  MoveC 2658 to (-287.4, 215.34, -30) mm, rotated rx 180 ry 0 rz 0.01 deg; joints [34.37, -40.028, 93.325, -139.792, 61.018, 158.683] to (-287.36, 219.75, -30) mm, rotated rx -180 ry 0 rz 0.01 deg; joints [34.501, -39.911, 93.073, -139.606, 60.965, 158.515]
  MoveC 2659 to (-287.18, 224.12, -30) mm, rotated rx 180 ry 0 rz 0.01 deg; joints [34.632, -39.801, 92.835, -139.421, 60.919, 158.351] to (-289.23, 227.97, -30) mm, rotated rx 180 ry 0 rz 0.01 deg; joints [34.703, -39.613, 92.434, -139.269, 60.786, 158.156]
  MoveC 2660 to (-302.15, 245.09, -30) mm, rotated rx -180 ry 0 rz 0.01 deg; joints [34.939, -38.61, 90.306, -138.602, 60.033, 157.181] to (-311.06, 264.6, -30) mm, rotated rx 180 ry 0 rz 0.01 deg; joints [35.316, -37.679, 88.333, -137.799, 59.413, 156.172]
  MoveC 2661 to (-313.16, 267.48, -30) mm, rotated rx -180 ry 0 rz 0.01 deg; joints [35.355, -37.507, 87.968, -137.682, 59.287, 156] to (-316.55, 268.57, -30) mm, rotated rx 180 ry 0 rz 0.01 deg; joints [35.318, -37.331, 87.599, -137.643, 59.129, 155.869]
  MoveL 2662 to (-329.31, 268.57, -30) mm, rotated rx 180 ry 0 rz 0.01 deg; joints [35.065, -36.784, 86.459, -137.668, 58.581, 155.543]
  MoveC 2663 to (-332.03, 267.45, -30) mm, rotated rx 180 ry 0 rz 0.01 deg; joints [34.98, -36.7, 86.285, -137.721, 58.477, 155.52] to (-333.16, 264.72, -30) mm, rotated rx 180 ry 0 rz 0.01 deg; joints [34.881, -36.731, 86.354, -137.84, 58.463, 155.605]
  MoveL 2664 to (-333.15, 129.67, -30) mm, rotated rx -180 ry 0 rz 0.01 deg; joints [30.91, -40.332, 94.104, -143.652, 60.117, 160.875]
  MoveC 2665 to (-332.02, 125.86, -30) mm, rotated rx -180 ry 0 rz 0.01 deg; joints [30.814, -40.47, 94.4, -143.81, 60.211, 161.035] to (-328.98, 123.31, -30) mm, rotated rx 180 ry 0 rz 0.01 deg; joints [30.791, -40.656, 94.796, -143.905, 60.373, 161.19]
  MoveC 2666 to (-314.64, 115.76, -30) mm, rotated rx 180 ry 0 rz 0.01 deg; joints [30.822, -41.42, 96.418, -144.154, 61.078, 161.751] to (-301.61, 106.12, -30) mm, rotated rx -180 ry 0 rz 0.01 deg; joints [30.764, -42.166, 98.01, -144.486, 61.745, 162.344]
  MoveC 2667 to (-290.27, 94.52, -30) mm, rotated rx -180 ry 0 rz 0.01 deg; joints [30.609, -42.877, 99.534, -144.901, 62.359, 162.955] to (-281.02, 81.2, -30) mm, rotated rx 180 ry 0 rz 0.01 deg; joints [30.356, -43.533, 100.948, -145.396, 62.903, 163.57]
  MoveL 2668 to (-263.17, 49.55, -30) mm, rotated rx 180 ry 0 rz 0.01 deg; joints [29.657, -44.892, 103.897, -146.586, 64.014, 164.905]
  MoveC 2669 to (-262.35, 48.05, -30) mm, rotated rx -180 ry 0 rz 0.01 deg; joints [29.623, -44.954, 104.032, -146.643, 64.065, 164.966] to (-261.62, 46.51, -30) mm, rotated rx -180 ry 0 rz 0.01 deg; joints [29.585, -45.014, 104.161, -146.702, 64.114, 165.027]
  MoveC 2670 to (-260.93, 44.95, -30) mm, rotated rx 180 ry 0 rz 0.01 deg; joints [29.546, -45.072, 104.289, -146.762, 64.16, 165.088] to (-260.22, 43.39, -30) mm, rotated rx -180 ry 0 rz 0.01 deg; joints [29.508, -45.131, 104.417, -146.821, 64.208, 165.148]
  MoveC 2671 to (-257.67, 40.46, -30) mm, rotated rx -180 ry 0 rz 0.01 deg; joints [29.458, -45.287, 104.757, -146.922, 64.347, 165.283] to (-253.93, 39.36, -30) mm, rotated rx -180 ry 0 rz 0.01 deg; joints [29.492, -45.45, 105.107, -146.935, 64.514, 165.38]
  MoveL 2672 to (-139.56, 39.36, -30) mm, rotated rx -180 ry 0 rz 0.01 deg; joints [31.818, -49.526, 113.886, -145.611, 69.031, 167.233]
  MoveC 2673 to (-135.82, 40.46, -30) mm, rotated rx 180 ry 0 rz 0.01 deg; joints [31.938, -49.631, 114.111, -145.512, 69.16, 167.26] to (-133.27, 43.42, -30) mm, rotated rx 180 ry 0 rz 0.01 deg; joints [32.098, -49.657, 114.162, -145.351, 69.219, 167.214]
  MoveC 2674 to (-132.52, 45.08, -30) mm, rotated rx 180 ry 0 rz 0.01 deg; joints [32.173, -49.649, 114.141, -145.271, 69.227, 167.178] to (-131.78, 46.75, -30) mm, rotated rx 180 ry 0 rz 0.01 deg; joints [32.247, -49.64, 114.118, -145.191, 69.234, 167.141]
  MoveC 2675 to (-131.01, 48.4, -30) mm, rotated rx -180 ry 0 rz 0.01 deg; joints [32.322, -49.633, 114.099, -145.11, 69.242, 167.106] to (-130.14, 50, -30) mm, rotated rx -180 ry 0 rz 0.01 deg; joints [32.397, -49.629, 114.088, -145.031, 69.255, 167.073]
  MoveL 2676 to (-112.26, 81.56, -30) mm, rotated rx -180 ry 0 rz 0.01 deg; joints [33.893, -49.569, 113.893, -143.455, 69.523, 166.428]
  MoveC 2677 to (-103.05, 94.8, -30) mm, rotated rx 180 ry 0 rz 0.01 deg; joints [34.56, -49.588, 113.908, -142.767, 69.693, 166.179] to (-91.75, 106.32, -30) mm, rotated rx 180 ry 0 rz 0.01 deg; joints [35.217, -49.706, 114.14, -142.117, 69.958, 166.013]
  MoveC 2678 to (-78.77, 115.88, -30) mm, rotated rx 180 ry 0 rz 0.01 deg; joints [35.853, -49.913, 114.573, -141.516, 70.303, 165.933] to (-64.48, 123.34, -30) mm, rotated rx 180 ry 0 rz 0.01 deg; joints [36.455, -50.202, 115.186, -140.973, 70.717, 165.937]
  MoveC 2679 to (-61.48, 125.84, -30) mm, rotated rx 180 ry 0 rz 0.01 deg; joints [36.613, -50.24, 115.265, -140.82, 70.791, 165.909] to (-60.36, 129.58, -30) mm, rotated rx 180 ry 0 rz 0.01 deg; joints [36.767, -50.191, 115.151, -140.649, 70.781, 165.812]
  MoveL 2680 to (-60.36, 264.73, -30) mm, rotated rx -180 ry 0 rz 0.01 deg; joints [41.026, -46.847, 107.689, -135.318, 69.022, 161.344]
  MoveC 2681 to (-61.49, 267.45, -30) mm, rotated rx 180 ry 0 rz 0.01 deg; joints [41.077, -46.737, 107.45, -135.232, 68.948, 161.227] to (-64.21, 268.58, -30) mm, rotated rx 180 ry 0 rz 0.01 deg; joints [41.041, -46.62, 107.197, -135.232, 68.838, 161.138]
  MoveL 2682 to (-76.96, 268.58, -30) mm, rotated rx 180 ry 0 rz 0.01 deg; joints [40.715, -46.209, 106.319, -135.431, 68.393, 160.909]
  MoveC 2683 to (-80.35, 267.48, -30) mm, rotated rx -180 ry 0 rz 0.01 deg; joints [40.597, -46.129, 106.149, -135.525, 68.288, 160.886] to (-82.45, 264.61, -30) mm, rotated rx -180 ry 0 rz 0.01 deg; joints [40.459, -46.138, 106.174, -135.668, 68.25, 160.951]
  MoveC 2684 to (-94.52, 240.3, -30) mm, rotated rx -180 ry 0 rz 0.01 deg; joints [39.431, -46.39, 106.752, -136.798, 68.133, 161.591] to (-112.91, 220.34, -30) mm, rotated rx -180 ry 0 rz 0.01 deg; joints [38.375, -46.299, 106.59, -137.853, 67.726, 161.954]
  MoveC 2685 to (-135.88, 205.99, -30) mm, rotated rx 180 ry 0 rz 0.01 deg; joints [37.386, -45.887, 105.736, -138.74, 67.068, 162.034] to (-161.71, 197.84, -30) mm, rotated rx -180 ry 0 rz 0.01 deg; joints [36.537, -45.199, 104.282, -139.395, 66.206, 161.843]
  MoveC 2686 to (-174.93, 196.15, -30) mm, rotated rx 180 ry 0 rz 0.01 deg; joints [36.185, -44.775, 103.382, -139.62, 65.727, 161.656] to (-188.26, 195.83, -30) mm, rotated rx 180 ry 0 rz 0.01 deg; joints [35.878, -44.307, 102.387, -139.783, 65.221, 161.417]
  MoveC 2687 to (-201.58, 196.1, -30) mm, rotated rx 180 ry 0 rz 0.01 deg; joints [35.593, -43.817, 101.348, -139.912, 64.703, 161.154] to (-214.9, 196.19, -30) mm, rotated rx -180 ry 0 rz 0.01 deg; joints [35.307, -43.325, 100.306, -140.04, 64.182, 160.893]
  MoveC 2688 to (-245.9, 200.97, -30) mm, rotated rx 180 ry 0 rz 0.01 deg; joints [34.794, -42.036, 97.572, -140.115, 62.891, 160.102] to (-274.04, 214.84, -30) mm, rotated rx 180 ry 0 rz 0.01 deg; joints [34.626, -40.576, 94.475, -139.736, 61.577, 158.995]
  MoveC 2689 to (-281.97, 221.02, -30) mm, rotated rx 180 ry 0 rz 0.01 deg; joints [34.647, -40.094, 93.454, -139.523, 61.173, 158.586] to (-289.23, 227.97, -30) mm, rotated rx 180 ry 0 rz 0.01 deg; joints [34.703, -39.613, 92.434, -139.269, 60.786, 158.156]
  MoveC 2690 to (-291.33, 232.25, -30) mm, rotated rx -180 ry 0 rz 0.01 deg; joints [34.785, -39.411, 92.003, -139.099, 60.646, 157.941] to (-290.67, 236.97, -30) mm, rotated rx 180 ry 0 rz 0.01 deg; joints [34.936, -39.307, 91.78, -138.897, 60.615, 157.771]
  MoveC 2691 to (-289.84, 241.61, -30) mm, rotated rx -180 ry 0 rz 0.01 deg; joints [35.087, -39.213, 91.574, -138.697, 60.592, 157.608] to (-291.43, 246.05, -30) mm, rotated rx -180 ry 0 rz 0.01 deg; joints [35.182, -39.024, 91.172, -138.517, 60.47, 157.395]
  MoveC 2692 to (-298.95, 259.4, -30) mm, rotated rx 180 ry 0 rz 0.01 deg; joints [35.412, -38.336, 89.712, -137.981, 59.989, 156.681] to (-303.93, 273.9, -30) mm, rotated rx -180 ry 0 rz 0.01 deg; joints [35.721, -37.707, 88.377, -137.381, 59.598, 155.964]
  MoveC 2693 to (-305.81, 276.81, -30) mm, rotated rx -180 ry 0 rz 0.01 deg; joints [35.765, -37.543, 88.029, -137.262, 59.482, 155.797] to (-309.08, 277.94, -30) mm, rotated rx 180 ry 0 rz 0.01 deg; joints [35.73, -37.371, 87.669, -137.222, 59.329, 155.667]
  MoveL 2694 to (-338.67, 277.94, -30) mm, rotated rx 180 ry 0 rz 0.01 deg; joints [35.143, -36.096, 85.013, -137.269, 58.056, 154.896]
  MoveC 2695 to (-341.39, 276.81, -30) mm, rotated rx -180 ry 0 rz 0.01 deg; joints [35.058, -36.01, 84.836, -137.32, 57.951, 154.872] to (-342.52, 274.08, -30) mm, rotated rx -180 ry 0 rz 0.01 deg; joints [34.96, -36.043, 84.907, -137.44, 57.936, 154.959]
  MoveL 2696 to (-342.52, 123.04, -30) mm, rotated rx -180 ry 0 rz 0.01 deg; joints [30.536, -40.1, 93.628, -143.974, 59.789, 160.915]
  MoveC 2697 to (-341.43, 119.51, -30) mm, rotated rx -180 ry 0 rz 0.01 deg; joints [30.447, -40.229, 93.906, -144.121, 59.878, 161.066] to (-338.54, 117.21, -30) mm, rotated rx 180 ry 0 rz 0.01 deg; joints [30.428, -40.404, 94.278, -144.208, 60.031, 161.209]
  MoveC 2698 to (-329.79, 113.4, -30) mm, rotated rx 180 ry 0 rz 0.01 deg; joints [30.469, -40.856, 95.234, -144.332, 60.456, 161.526] to (-321.33, 108.99, -30) mm, rotated rx -180 ry 0 rz 0.01 deg; joints [30.487, -41.305, 96.188, -144.478, 60.872, 161.853]
  MoveC 2699 to (-313.31, 103.8, -30) mm, rotated rx 180 ry 0 rz 0.01 deg; joints [30.472, -41.75, 97.135, -144.654, 61.276, 162.194] to (-305.96, 97.7, -30) mm, rotated rx -180 ry 0 rz 0.01 deg; joints [30.416, -42.184, 98.062, -144.87, 61.66, 162.547]
  MoveC 2700 to (-295.26, 85.95, -30) mm, rotated rx 180 ry 0 rz 0.01 deg; joints [30.241, -42.872, 99.537, -145.298, 62.251, 163.148] to (-286.59, 72.62, -30) mm, rotated rx -180 ry 0 rz 0.01 deg; joints [29.974, -43.503, 100.899, -145.8, 62.771, 163.749]
  MoveL 2701 to (-271.14, 44.96, -30) mm, rotated rx -180 ry 0 rz 0.01 deg; joints [29.355, -44.683, 103.46, -146.848, 63.738, 164.911]
  MoveC 2702 to (-269.76, 42.31, -30) mm, rotated rx -180 ry 0 rz 0.01 deg; joints [29.292, -44.79, 103.693, -146.949, 63.826, 165.018] to (-268.6, 39.56, -30) mm, rotated rx 180 ry 0 rz 0.01 deg; joints [29.222, -44.891, 103.913, -147.055, 63.907, 165.124]
  MoveC 2703 to (-267.53, 36.78, -30) mm, rotated rx -180 ry 0 rz 0.01 deg; joints [29.149, -44.988, 104.126, -147.164, 63.983, 165.229] to (-266.4, 34.01, -30) mm, rotated rx -180 ry 0 rz 0.01 deg; joints [29.078, -45.087, 104.342, -147.271, 64.062, 165.334]
  MoveC 2704 to (-263.99, 31.09, -30) mm, rotated rx -180 ry 0 rz 0.01 deg; joints [29.025, -45.237, 104.669, -147.374, 64.196, 165.465] to (-260.37, 30, -30) mm, rotated rx 180 ry 0 rz 0.01 deg; joints [29.056, -45.396, 105.01, -147.389, 64.358, 165.56]
  MoveL 2705 to (-133.13, 30, -30) mm, rotated rx -180 ry 0 rz 0.01 deg; joints [31.628, -49.928, 114.781, -145.913, 69.393, 167.601]
  MoveC 2706 to (-129.52, 31.09, -30) mm, rotated rx 180 ry 0 rz 0.01 deg; joints [31.745, -50.028, 114.996, -145.815, 69.516, 167.626] to (-127.12, 33.98, -30) mm, rotated rx 180 ry 0 rz 0.01 deg; joints [31.901, -50.051, 115.04, -145.659, 69.571, 167.581]
  MoveC 2707 to (-125.94, 36.86, -30) mm, rotated rx 180 ry 0 rz 0.01 deg; joints [32.029, -50.033, 114.995, -145.52, 69.579, 167.517] to (-124.82, 39.77, -30) mm, rotated rx -180 ry 0 rz 0.01 deg; joints [32.156, -50.013, 114.944, -145.382, 69.584, 167.451]
  MoveC 2708 to (-123.61, 42.64, -30) mm, rotated rx 180 ry 0 rz 0.01 deg; joints [32.284, -49.996, 114.901, -145.244, 69.594, 167.388] to (-122.17, 45.4, -30) mm, rotated rx -180 ry 0 rz 0.01 deg; joints [32.413, -49.988, 114.879, -145.107, 69.613, 167.331]
  MoveL 2709 to (-103.15, 78.32, -30) mm, rotated rx 180 ry 0 rz 0.01 deg; joints [33.993, -49.937, 114.701, -143.449, 69.902, 166.67]
  MoveC 2710 to (-91.63, 93.87, -30) mm, rotated rx -180 ry 0 rz 0.01 deg; joints [34.797, -49.981, 114.763, -142.626, 70.123, 166.391] to (-76.92, 106.43, -30) mm, rotated rx 180 ry 0 rz 0.01 deg; joints [35.578, -50.181, 115.174, -141.871, 70.493, 166.25]
  MoveC 2711 to (-71.7, 109.64, -30) mm, rotated rx 180 ry 0 rz 0.01 deg; joints [35.814, -50.277, 115.377, -141.653, 70.638, 166.237] to (-66.23, 112.38, -30) mm, rotated rx 180 ry 0 rz 0.01 deg; joints [36.042, -50.39, 115.619, -141.448, 70.798, 166.242]
  MoveC 2712 to (-60.63, 114.83, -30) mm, rotated rx 180 ry 0 rz 0.01 deg; joints [36.263, -50.513, 115.882, -141.252, 70.966, 166.258] to (-54.97, 117.16, -30) mm, rotated rx 180 ry 0 rz 0.01 deg; joints [36.483, -50.639, 116.152, -141.059, 71.136, 166.279]
  MoveC 2713 to (-52.08, 119.49, -30) mm, rotated rx 180 ry 0 rz 0.01 deg; joints [36.635, -50.678, 116.232, -140.913, 71.207, 166.255] to (-50.99, 123.04, -30) mm, rotated rx 180 ry 0 rz 0.01 deg; joints [36.782, -50.632, 116.126, -140.75, 71.198, 166.164]
  MoveL 2714 to (-51, 274.09, -30) mm, rotated rx 180 ry 0 rz 0.01 deg; joints [41.545, -46.89, 107.767, -134.806, 69.225, 161.178]
  MoveC 2715 to (-52.13, 276.81, -30) mm, rotated rx 180 ry 0 rz 0.01 deg; joints [41.596, -46.781, 107.527, -134.72, 69.151, 161.061] to (-54.85, 277.94, -30) mm, rotated rx 180 ry 0 rz 0.01 deg; joints [41.558, -46.663, 107.275, -134.721, 69.043, 160.972]
  MoveL 2716 to (-84.48, 277.94, -30) mm, rotated rx -180 ry 0 rz 0.01 deg; joints [40.8, -45.709, 105.236, -135.182, 68.009, 160.435]
  MoveC 2717 to (-87.74, 276.81, -30) mm, rotated rx -180 ry 0 rz 0.01 deg; joints [40.684, -45.633, 105.077, -135.274, 67.908, 160.416] to (-89.59, 273.9, -30) mm, rotated rx 180 ry 0 rz 0.01 deg; joints [40.553, -45.652, 105.121, -135.414, 67.879, 160.487]
  MoveC 2718 to (-96.46, 255.09, -30) mm, rotated rx 180 ry 0 rz 0.01 deg; joints [39.826, -45.935, 105.754, -136.247, 67.875, 161.035] to (-107.51, 238.41, -30) mm, rotated rx -180 ry 0 rz 0.01 deg; joints [39.054, -46.01, 105.942, -137.062, 67.691, 161.423]
  MoveC 2719 to (-122.04, 224.65, -30) mm, rotated rx -180 ry 0 rz 0.01 deg; joints [38.286, -45.881, 105.689, -137.809, 67.339, 161.64] to (-139.21, 214.4, -30) mm, rotated rx 180 ry 0 rz 0.01 deg; joints [37.566, -45.56, 105.022, -138.447, 66.838, 161.683]
  MoveC 2720 to (-148.66, 210.65, -30) mm, rotated rx 180 ry 0 rz 0.01 deg; joints [37.231, -45.33, 104.538, -138.719, 66.534, 161.64] to (-158.44, 207.86, -30) mm, rotated rx 180 ry 0 rz 0.01 deg; joints [36.919, -45.06, 103.969, -138.952, 66.204, 161.556]
  MoveC 2721 to (-168.46, 206.14, -30) mm, rotated rx -180 ry 0 rz 0.01 deg; joints [36.638, -44.752, 103.316, -139.141, 65.847, 161.429] to (-178.62, 205.56, -30) mm, rotated rx -180 ry 0 rz 0.01 deg; joints [36.391, -44.406, 102.582, -139.281, 65.469, 161.259]
  MoveL 2722 to (-217.27, 205.67, -30) mm, rotated rx -180 ry 0 rz 0.01 deg; joints [35.543, -42.995, 99.591, -139.675, 63.971, 160.508]
  MoveC 2723 to (-236.59, 208, -30) mm, rotated rx 180 ry 0 rz 0.01 deg; joints [35.201, -42.209, 97.926, -139.749, 63.177, 160.035] to (-254.87, 214.67, -30) mm, rotated rx 180 ry 0 rz 0.01 deg; joints [35.016, -41.332, 96.068, -139.615, 62.361, 159.411]
  MoveC 2724 to (-271.59, 225.24, -30) mm, rotated rx 180 ry 0 rz 0.01 deg; joints [34.983, -40.394, 94.078, -139.286, 61.549, 158.654] to (-285.91, 238.89, -30) mm, rotated rx -180 ry 0 rz 0.01 deg; joints [35.088, -39.448, 92.07, -138.792, 60.789, 157.805]
  MoveC 2725 to (-288.76, 242.4, -30) mm, rotated rx 180 ry 0 rz 0.01 deg; joints [35.131, -39.235, 91.618, -138.658, 60.627, 157.602] to (-291.43, 246.05, -30) mm, rotated rx -180 ry 0 rz 0.01 deg; joints [35.182, -39.024, 91.172, -138.517, 60.47, 157.395]
  MoveC 2726 to (-292.73, 250.22, -30) mm, rotated rx -180 ry 0 rz 0.01 deg; joints [35.276, -38.853, 90.808, -138.346, 60.364, 157.199] to (-291.43, 254.39, -30) mm, rotated rx 180 ry 0 rz 0.01 deg; joints [35.421, -38.788, 90.666, -138.164, 60.366, 157.062]
  MoveC 2727 to (-289.96, 258.45, -30) mm, rotated rx 180 ry 0 rz 0.01 deg; joints [35.567, -38.733, 90.544, -137.986, 60.377, 156.934] to (-290.67, 262.7, -30) mm, rotated rx 180 ry 0 rz 0.01 deg; joints [35.674, -38.582, 90.222, -137.809, 60.294, 156.746]
  MoveC 2728 to (-292.97, 268.55, -30) mm, rotated rx 180 ry 0 rz 0.01 deg; joints [35.793, -38.319, 89.662, -137.57, 60.125, 156.453] to (-294.74, 274.58, -30) mm, rotated rx 180 ry 0 rz 0.01 deg; joints [35.927, -38.07, 89.133, -137.321, 59.975, 156.162]
  MoveC 2729 to (-295.23, 276.75, -30) mm, rotated rx -180 ry 0 rz 0.01 deg; joints [35.978, -37.986, 88.955, -137.23, 59.928, 156.061] to (-295.64, 278.92, -30) mm, rotated rx 180 ry 0 rz 0.01 deg; joints [36.031, -37.905, 88.782, -137.139, 59.883, 155.961]
  MoveC 2730 to (-296.04, 281.1, -30) mm, rotated rx 180 ry 0 rz 0.01 deg; joints [36.084, -37.824, 88.61, -137.048, 59.839, 155.861] to (-296.5, 283.27, -30) mm, rotated rx -180 ry 0 rz 0.01 deg; joints [36.135, -37.741, 88.433, -136.957, 59.793, 155.759]
  MoveC 2731 to (-298.31, 286.17, -30) mm, rotated rx -180 ry 0 rz 0.01 deg; joints [36.179, -37.579, 88.091, -136.839, 59.68, 155.593] to (-301.53, 287.3, -30) mm, rotated rx 180 ry 0 rz 0.01 deg; joints [36.145, -37.41, 87.737, -136.8, 59.53, 155.465]
  MoveL 2732 to (-348.03, 287.3, -30) mm, rotated rx -180 ry 0 rz 0.01 deg; joints [35.219, -35.396, 83.542, -136.858, 57.526, 154.232]
  MoveC 2733 to (-350.76, 286.17, -30) mm, rotated rx 180 ry 0 rz 0.01 deg; joints [35.135, -35.308, 83.362, -136.906, 57.421, 154.206] to (-351.88, 283.45, -30) mm, rotated rx 180 ry 0 rz 0.01 deg; joints [35.038, -35.342, 83.435, -137.026, 57.405, 154.295]
  MoveL 2734 to (-351.88, 115.54, -30) mm, rotated rx -180 ry 0 rz 0.01 deg; joints [30.136, -39.884, 93.188, -144.331, 59.468, 160.987]
  MoveC 2735 to (-350.79, 112.34, -30) mm, rotated rx 180 ry 0 rz 0.01 deg; joints [30.057, -40.006, 93.449, -144.465, 59.553, 161.125] to (-347.98, 110.47, -30) mm, rotated rx 180 ry 0 rz 0.01 deg; joints [30.049, -40.168, 93.793, -144.535, 59.699, 161.252]
  MoveC 2736 to (-334.23, 105.41, -30) mm, rotated rx 180 ry 0 rz 0.01 deg; joints [30.14, -40.859, 95.254, -144.694, 60.358, 161.717] to (-321.65, 97.91, -30) mm, rotated rx 180 ry 0 rz 0.01 deg; joints [30.133, -41.546, 96.715, -144.952, 60.988, 162.232]
  MoveC 2737 to (-310.51, 88.44, -30) mm, rotated rx 180 ry 0 rz 0.01 deg; joints [30.038, -42.209, 98.132, -145.291, 61.576, 162.774] to (-300.91, 77.41, -30) mm, rotated rx 180 ry 0 rz 0.01 deg; joints [29.862, -42.836, 99.477, -145.698, 62.112, 163.326]
  MoveL 2738 to (-279.12, 40.36, -30) mm, rotated rx -180 ry 0 rz 0.01 deg; joints [29.054, -44.471, 103.017, -147.108, 63.46, 164.918]
  MoveC 2739 to (-277.19, 36.6, -30) mm, rotated rx 180 ry 0 rz 0.01 deg; joints [28.964, -44.622, 103.346, -147.252, 63.584, 165.069] to (-275.65, 32.66, -30) mm, rotated rx -180 ry 0 rz 0.01 deg; joints [28.861, -44.761, 103.65, -147.406, 63.693, 165.218]
  MoveC 2740 to (-274.29, 28.67, -30) mm, rotated rx 180 ry 0 rz 0.01 deg; joints [28.753, -44.894, 103.94, -147.565, 63.796, 165.365] to (-272.91, 24.68, -30) mm, rotated rx -180 ry 0 rz 0.01 deg; joints [28.644, -45.026, 104.23, -147.722, 63.9, 165.512]
  MoveC 2741 to (-270.71, 21.75, -30) mm, rotated rx -180 ry 0 rz 0.01 deg; joints [28.586, -45.168, 104.54, -147.828, 64.025, 165.639] to (-267.22, 20.64, -30) mm, rotated rx 180 ry 0 rz 0.01 deg; joints [28.613, -45.323, 104.873, -147.846, 64.183, 165.732]
  MoveL 2742 to (-126.29, 20.64, -30) mm, rotated rx -180 ry 0 rz 0.01 deg; joints [31.444, -50.34, 115.699, -146.209, 69.77, 167.972]
  MoveC 2743 to (-122.81, 21.75, -30) mm, rotated rx 180 ry 0 rz 0.01 deg; joints [31.56, -50.435, 115.904, -146.111, 69.888, 167.994] to (-120.6, 24.67, -30) mm, rotated rx 180 ry 0 rz 0.01 deg; joints [31.713, -50.451, 115.933, -145.955, 69.934, 167.946]
  MoveC 2744 to (-119.17, 28.77, -30) mm, rotated rx -180 ry 0 rz 0.01 deg; joints [31.891, -50.418, 115.853, -145.761, 69.936, 167.852] to (-117.77, 32.88, -30) mm, rotated rx -180 ry 0 rz 0.01 deg; joints [32.069, -50.384, 115.769, -145.567, 69.937, 167.757]
  MoveC 2745 to (-116.18, 36.92, -30) mm, rotated rx -180 ry 0 rz 0.01 deg; joints [32.248, -50.356, 115.7, -145.373, 69.946, 167.667] to (-114.2, 40.79, -30) mm, rotated rx -180 ry 0 rz 0.01 deg; joints [32.429, -50.345, 115.667, -145.181, 69.971, 167.588]
  MoveL 2746 to (-96.23, 72.15, -30) mm, rotated rx -180 ry 0 rz 0.01 deg; joints [33.941, -50.292, 115.487, -143.596, 70.235, 166.962]
  MoveC 2747 to (-85.49, 86.83, -30) mm, rotated rx 180 ry 0 rz 0.01 deg; joints [34.702, -50.33, 115.539, -142.816, 70.438, 166.699] to (-71.68, 98.67, -30) mm, rotated rx -180 ry 0 rz 0.01 deg; joints [35.441, -50.517, 115.924, -142.101, 70.783, 166.567]
  MoveC 2748 to (-65.54, 102.43, -30) mm, rotated rx -180 ry 0 rz 0.01 deg; joints [35.72, -50.63, 116.163, -141.842, 70.954, 166.553] to (-59.09, 105.64, -30) mm, rotated rx 180 ry 0 rz 0.01 deg; joints [35.989, -50.764, 116.448, -141.6, 71.141, 166.56]
  MoveC 2749 to (-52.41, 108.31, -30) mm, rotated rx -180 ry 0 rz 0.01 deg; joints [36.247, -50.915, 116.773, -141.373, 71.344, 166.587] to (-45.54, 110.47, -30) mm, rotated rx 180 ry 0 rz 0.01 deg; joints [36.493, -51.081, 117.134, -141.163, 71.557, 166.633]
  MoveC 2750 to (-42.72, 112.37, -30) mm, rotated rx -180 ry 0 rz 0.01 deg; joints [36.629, -51.127, 117.229, -141.035, 71.631, 166.621] to (-41.63, 115.59, -30) mm, rotated rx -180 ry 0 rz 0.01 deg; joints [36.766, -51.089, 117.141, -140.884, 71.627, 166.541]
  MoveL 2751 to (-41.63, 283.45, -30) mm, rotated rx 180 ry 0 rz 0.01 deg; joints [42.066, -46.929, 107.834, -134.292, 69.425, 161.011]
  MoveC 2752 to (-42.76, 286.18, -30) mm, rotated rx -180 ry 0 rz 0.01 deg; joints [42.115, -46.818, 107.594, -134.207, 69.352, 160.893] to (-45.49, 287.31, -30) mm, rotated rx -180 ry 0 rz 0.01 deg; joints [42.076, -46.702, 107.342, -134.209, 69.244, 160.804]
  MoveL 2753 to (-91.92, 287.31, -30) mm, rotated rx -180 ry 0 rz 0.01 deg; joints [40.885, -45.205, 104.148, -134.928, 67.626, 159.956]
  MoveC 2754 to (-95.15, 286.18, -30) mm, rotated rx -180 ry 0 rz 0.01 deg; joints [40.772, -45.13, 103.989, -135.017, 67.525, 159.937] to (-96.98, 283.3, -30) mm, rotated rx 180 ry 0 rz 0.01 deg; joints [40.642, -45.149, 104.035, -135.155, 67.497, 160.008]
  MoveL 2755 to (-99.67, 271.79, -30) mm, rotated rx -180 ry 0 rz 0.01 deg; joints [40.24, -45.377, 104.538, -135.642, 67.547, 160.377]
  MoveC 2756 to (-101.4, 266.12, -30) mm, rotated rx -180 ry 0 rz 0.01 deg; joints [40.03, -45.474, 104.753, -135.887, 67.558, 160.549] to (-103.9, 260.75, -30) mm, rotated rx 180 ry 0 rz 0.01 deg; joints [39.81, -45.536, 104.894, -136.133, 67.536, 160.696]
  MoveC 2757 to (-115.59, 244.22, -30) mm, rotated rx -180 ry 0 rz 0.01 deg; joints [39.032, -45.586, 105.029, -136.946, 67.325, 161.07] to (-130.59, 230.61, -30) mm, rotated rx -180 ry 0 rz 0.01 deg; joints [38.262, -45.436, 104.731, -137.688, 66.951, 161.274]
  MoveC 2758 to (-148.37, 220.85, -30) mm, rotated rx 180 ry 0 rz 0.01 deg; joints [37.548, -45.078, 103.985, -138.306, 66.417, 161.288] to (-168.02, 215.81, -30) mm, rotated rx 180 ry 0 rz 0.01 deg; joints [36.942, -44.52, 102.806, -138.746, 65.743, 161.097]
  MoveC 2759 to (-170.66, 215.49, -30) mm, rotated rx -180 ry 0 rz 0.01 deg; joints [36.872, -44.434, 102.625, -138.789, 65.647, 161.059] to (-173.31, 215.2, -30) mm, rotated rx -180 ry 0 rz 0.01 deg; joints [36.804, -44.348, 102.442, -138.831, 65.55, 161.019]
  MoveC 2760 to (-175.96, 214.99, -30) mm, rotated rx 180 ry 0 rz 0.01 deg; joints [36.737, -44.259, 102.254, -138.87, 65.452, 160.976] to (-178.62, 214.92, -30) mm, rotated rx 180 ry 0 rz 0.01 deg; joints [36.675, -44.166, 102.056, -138.902, 65.352, 160.928]
  MoveL 2761 to (-215.12, 214.78, -30) mm, rotated rx 180 ry 0 rz 0.01 deg; joints [35.864, -42.839, 99.246, -139.281, 63.943, 160.221]
  MoveC 2762 to (-233.39, 216.8, -30) mm, rotated rx 180 ry 0 rz 0.01 deg; joints [35.532, -42.101, 97.683, -139.359, 63.196, 159.778] to (-250.67, 223.04, -30) mm, rotated rx 180 ry 0 rz 0.01 deg; joints [35.352, -41.273, 95.929, -139.237, 62.427, 159.187]
  MoveC 2763 to (-265.48, 232.24, -30) mm, rotated rx 180 ry 0 rz 0.01 deg; joints [35.314, -40.447, 94.177, -138.955, 61.712, 158.52] to (-278.37, 243.97, -30) mm, rotated rx 180 ry 0 rz 0.01 deg; joints [35.389, -39.611, 92.405, -138.54, 61.038, 157.778]
  MoveC 2764 to (-285.28, 252.84, -30) mm, rotated rx 180 ry 0 rz 0.01 deg; joints [35.503, -39.083, 91.286, -138.201, 60.642, 157.269] to (-290.67, 262.7, -30) mm, rotated rx 180 ry 0 rz 0.01 deg; joints [35.674, -38.582, 90.222, -137.809, 60.294, 156.746]
  MoveC 2765 to (-291.21, 267.33, -30) mm, rotated rx 180 ry 0 rz 0.01 deg; joints [35.794, -38.427, 89.89, -137.615, 60.214, 156.545] to (-289, 271.43, -30) mm, rotated rx 180 ry 0 rz 0.01 deg; joints [35.955, -38.399, 89.826, -137.432, 60.255, 156.431]
  MoveC 2766 to (-286.63, 275.37, -30) mm, rotated rx 180 ry 0 rz 0.01 deg; joints [36.115, -38.381, 89.783, -137.256, 60.304, 156.327] to (-286.52, 279.96, -30) mm, rotated rx 180 ry 0 rz 0.01 deg; joints [36.247, -38.252, 89.505, -137.061, 60.251, 156.142]
  MoveC 2767 to (-287.85, 286.38, -30) mm, rotated rx 180 ry 0 rz 0.01 deg; joints [36.399, -38.007, 88.985, -136.794, 60.115, 155.844] to (-288.78, 292.87, -30) mm, rotated rx 180 ry 0 rz 0.01 deg; joints [36.561, -37.776, 88.491, -136.522, 59.995, 155.551]
  MoveC 2768 to (-290.17, 295.58, -30) mm, rotated rx 180 ry 0 rz 0.01 deg; joints [36.608, -37.636, 88.196, -136.412, 59.902, 155.402] to (-293.02, 296.66, -30) mm, rotated rx 180 ry 0 rz 0.01 deg; joints [36.579, -37.485, 87.879, -136.375, 59.77, 155.285]
  MoveL 2769 to (-357.39, 296.66, -30) mm, rotated rx 180 ry 0 rz 0.01 deg; joints [35.295, -34.682, 82.045, -136.433, 56.992, 153.55]
  MoveC 2770 to (-360.12, 295.53, -30) mm, rotated rx 180 ry 0 rz 0.01 deg; joints [35.211, -34.593, 81.862, -136.479, 56.885, 153.521] to (-361.25, 292.81, -30) mm, rotated rx 180 ry 0 rz 0.01 deg; joints [35.115, -34.627, 81.937, -136.599, 56.869, 153.611]
  MoveL 2771 to (-361.24, 107.51, -30) mm, rotated rx -180 ry 0 rz 0.01 deg; joints [29.722, -39.677, 92.765, -144.708, 59.149, 161.076]
  MoveC 2772 to (-360.16, 104.51, -30) mm, rotated rx -180 ry 0 rz 0.01 deg; joints [29.649, -39.793, 93.015, -144.834, 59.232, 161.208] to (-357.4, 102.89, -30) mm, rotated rx -180 ry 0 rz 0.01 deg; joints [29.647, -39.948, 93.342, -144.895, 59.373, 161.324]
  MoveC 2773 to (-352.8, 101.95, -30) mm, rotated rx 180 ry 0 rz 0.01 deg; joints [29.699, -40.164, 93.798, -144.919, 59.587, 161.455] to (-348.24, 100.85, -30) mm, rotated rx -180 ry 0 rz 0.01 deg; joints [29.746, -40.381, 94.257, -144.95, 59.8, 161.589]
  MoveC 2774 to (-343.74, 99.49, -30) mm, rotated rx -180 ry 0 rz 0.01 deg; joints [29.784, -40.601, 94.721, -144.99, 60.013, 161.73] to (-339.36, 97.79, -30) mm, rotated rx -180 ry 0 rz 0.01 deg; joints [29.809, -40.822, 95.189, -145.044, 60.224, 161.88]
  MoveC 2775 to (-321.77, 86.74, -30) mm, rotated rx 180 ry 0 rz 0.01 deg; joints [29.778, -41.793, 97.256, -145.428, 61.114, 162.613] to (-308.28, 70.94, -30) mm, rotated rx -180 ry 0 rz 0.01 deg; joints [29.519, -42.683, 99.166, -146.02, 61.875, 163.403]
  MoveL 2776 to (-287.22, 35.69, -30) mm, rotated rx 180 ry 0 rz 0.01 deg; joints [28.75, -44.253, 102.563, -147.369, 63.174, 164.924]
  MoveC 2777 to (-284.73, 30.82, -30) mm, rotated rx -180 ry 0 rz 0.01 deg; joints [28.634, -44.448, 102.987, -147.557, 63.335, 165.119] to (-282.75, 25.72, -30) mm, rotated rx 180 ry 0 rz 0.01 deg; joints [28.499, -44.627, 103.378, -147.758, 63.477, 165.312]
  MoveC 2778 to (-281.17, 20.49, -30) mm, rotated rx -180 ry 0 rz 0.01 deg; joints [28.353, -44.792, 103.74, -147.967, 63.603, 165.501] to (-279.85, 15.19, -30) mm, rotated rx 180 ry 0 rz 0.01 deg; joints [28.198, -44.948, 104.082, -148.182, 63.719, 165.686]
  MoveC 2779 to (-278.1, 12.37, -30) mm, rotated rx -180 ry 0 rz 0.01 deg; joints [28.135, -45.071, 104.349, -148.288, 63.825, 165.802] to (-274.97, 11.27, -30) mm, rotated rx -180 ry 0 rz 0.01 deg; joints [28.154, -45.212, 104.653, -148.309, 63.968, 165.888]
  MoveL 2780 to (-118.61, 11.27, -30) mm, rotated rx 180 ry 0 rz 0.01 deg; joints [31.276, -50.775, 116.672, -146.492, 70.179, 168.35]
  MoveC 2781 to (-115.43, 12.39, -30) mm, rotated rx -180 ry 0 rz 0.01 deg; joints [31.386, -50.859, 116.853, -146.397, 70.285, 168.367] to (-113.65, 15.25, -30) mm, rotated rx 180 ry 0 rz 0.01 deg; joints [31.529, -50.863, 116.856, -146.249, 70.316, 168.315]
  MoveC 2782 to (-109.31, 29.24, -30) mm, rotated rx 180 ry 0 rz 0.01 deg; joints [32.128, -50.734, 116.543, -145.592, 70.301, 167.99] to (-102.79, 42.36, -30) mm, rotated rx -180 ry 0 rz 0.01 deg; joints [32.743, -50.688, 116.414, -144.94, 70.376, 167.72]
  MoveL 2783 to (-87.95, 67.51, -30) mm, rotated rx -180 ry 0 rz 0.01 deg; joints [33.973, -50.658, 116.294, -143.655, 70.599, 167.228]
  MoveC 2784 to (-80.44, 78.02, -30) mm, rotated rx 180 ry 0 rz 0.01 deg; joints [34.518, -50.679, 116.32, -143.097, 70.737, 167.04] to (-71.05, 86.89, -30) mm, rotated rx 180 ry 0 rz 0.01 deg; joints [35.051, -50.791, 116.545, -142.574, 70.96, 166.927]
  MoveC 2785 to (-60.38, 94.12, -30) mm, rotated rx -180 ry 0 rz 0.01 deg; joints [35.562, -50.973, 116.93, -142.094, 71.248, 166.883] to (-48.85, 99.87, -30) mm, rotated rx -180 ry 0 rz 0.01 deg; joints [36.046, -51.21, 117.437, -141.655, 71.581, 166.896]
  MoveC 2786 to (-45.65, 101, -30) mm, rotated rx 180 ry 0 rz 0.01 deg; joints [36.166, -51.285, 117.598, -141.551, 71.679, 166.913] to (-42.35, 101.77, -30) mm, rotated rx 180 ry 0 rz 0.01 deg; joints [36.276, -51.371, 117.785, -141.46, 71.786, 166.943]
  MoveL 2787 to (-36.21, 102.84, -30) mm, rotated rx 180 ry 0 rz 0.01 deg; joints [36.468, -51.537, 118.148, -141.304, 71.987, 167.009]
  MoveC 2788 to (-33.38, 104.46, -30) mm, rotated rx 180 ry 0 rz 0.01 deg; joints [36.596, -51.588, 118.258, -141.185, 72.064, 167.006] to (-32.27, 107.53, -30) mm, rotated rx 180 ry 0 rz 0.01 deg; joints [36.73, -51.555, 118.179, -141.04, 72.062, 166.933]
  MoveL 2789 to (-32.27, 292.82, -30) mm, rotated rx 180 ry 0 rz 0.01 deg; joints [42.586, -46.962, 107.891, -133.778, 69.623, 160.841]
  MoveC 2790 to (-33.4, 295.54, -30) mm, rotated rx -180 ry 0 rz 0.01 deg; joints [42.635, -46.851, 107.649, -133.694, 69.55, 160.722] to (-36.13, 296.67, -30) mm, rotated rx 180 ry 0 rz 0.01 deg; joints [42.595, -46.735, 107.399, -133.697, 69.443, 160.633]
  MoveL 2791 to (-100.53, 296.67, -30) mm, rotated rx 180 ry 0 rz 0.01 deg; joints [40.94, -44.658, 102.969, -134.686, 67.201, 159.449]
  MoveC 2792 to (-103.36, 295.58, -30) mm, rotated rx 180 ry 0 rz 0.01 deg; joints [40.838, -44.594, 102.834, -134.767, 67.113, 159.435] to (-104.73, 292.88, -30) mm, rotated rx 180 ry 0 rz 0.01 deg; joints [40.726, -44.624, 102.902, -134.891, 67.099, 159.509]
  MoveC 2793 to (-106.48, 282.44, -30) mm, rotated rx -180 ry 0 rz 0.01 deg; joints [40.382, -44.856, 103.413, -135.322, 67.168, 159.861] to (-109.53, 272.3, -30) mm, rotated rx -180 ry 0 rz 0.01 deg; joints [40.011, -45.034, 103.807, -135.759, 67.187, 160.175]
  MoveC 2794 to (-113.87, 262.64, -30) mm, rotated rx 180 ry 0 rz 0.01 deg; joints [39.621, -45.151, 104.071, -136.197, 67.153, 160.443] to (-119.51, 253.68, -30) mm, rotated rx 180 ry 0 rz 0.01 deg; joints [39.219, -45.202, 104.195, -136.627, 67.063, 160.661]
  MoveC 2795 to (-128.96, 243.24, -30) mm, rotated rx 180 ry 0 rz 0.01 deg; joints [38.681, -45.159, 104.121, -137.165, 66.85, 160.857] to (-140.39, 235.03, -30) mm, rotated rx 180 ry 0 rz 0.01 deg; joints [38.163, -44.984, 103.762, -137.639, 66.534, 160.936]
  MoveC 2796 to (-153.15, 229.14, -30) mm, rotated rx 180 ry 0 rz 0.01 deg; joints [37.687, -44.696, 103.159, -138.033, 66.134, 160.906] to (-166.71, 225.48, -30) mm, rotated rx 180 ry 0 rz 0.01 deg; joints [37.264, -44.315, 102.355, -138.341, 65.671, 160.779]
  MoveC 2797 to (-178.7, 223.98, -30) mm, rotated rx -180 ry 0 rz 0.01 deg; joints [36.947, -43.928, 101.536, -138.537, 65.235, 160.603] to (-190.78, 223.8, -30) mm, rotated rx -180 ry 0 rz 0.01 deg; joints [36.67, -43.497, 100.623, -138.674, 64.775, 160.375]
  MoveC 2798 to (-202.83, 224.16, -30) mm, rotated rx 180 ry 0 rz 0.01 deg; joints [36.413, -43.047, 99.671, -138.781, 64.305, 160.125] to (-214.9, 224.28, -30) mm, rotated rx 180 ry 0 rz 0.01 deg; joints [36.153, -42.598, 98.721, -138.89, 63.833, 159.879]
  MoveC 2799 to (-233.07, 226.62, -30) mm, rotated rx 180 ry 0 rz 0.01 deg; joints [35.83, -41.853, 97.145, -138.953, 63.087, 159.422] to (-250.06, 233.48, -30) mm, rotated rx 180 ry 0 rz 0.01 deg; joints [35.672, -41.017, 95.373, -138.8, 62.322, 158.807]
  MoveC 2800 to (-264.91, 244.15, -30) mm, rotated rx -180 ry 0 rz 0.01 deg; joints [35.672, -40.143, 93.521, -138.455, 61.588, 158.073] to (-277.02, 257.85, -30) mm, rotated rx 180 ry 0 rz 0.01 deg; joints [35.816, -39.276, 91.682, -137.95, 60.921, 157.261]
  MoveC 2801 to (-281.75, 265.9, -30) mm, rotated rx 180 ry 0 rz 0.01 deg; joints [35.948, -38.855, 90.788, -137.634, 60.625, 156.828] to (-285.1, 274.62, -30) mm, rotated rx 180 ry 0 rz 0.01 deg; joints [36.126, -38.466, 89.961, -137.281, 60.377, 156.395]
  MoveC 2802 to (-285.85, 277.28, -30) mm, rotated rx 180 ry 0 rz 0.01 deg; joints [36.185, -38.358, 89.731, -137.172, 60.313, 156.268] to (-286.52, 279.96, -30) mm, rotated rx -180 ry 0 rz 0.01 deg; joints [36.247, -38.252, 89.505, -137.061, 60.251, 156.142]
  MoveC 2803 to (-286.22, 284.31, -30) mm, rotated rx 180 ry 0 rz 0.01 deg; joints [36.375, -38.136, 89.256, -136.876, 60.209, 155.969] to (-283.5, 287.72, -30) mm, rotated rx 180 ry 0 rz 0.01 deg; joints [36.527, -38.147, 89.274, -136.72, 60.279, 155.895]
  MoveC 2804 to (-280.64, 290.93, -30) mm, rotated rx -180 ry 0 rz 0.01 deg; joints [36.676, -38.168, 89.314, -136.573, 60.357, 155.831] to (-279.69, 295.12, -30) mm, rotated rx -180 ry 0 rz 0.01 deg; joints [36.813, -38.082, 89.128, -136.392, 60.344, 155.681]
  MoveC 2805 to (-279.68, 298.76, -30) mm, rotated rx -180 ry 0 rz 0.01 deg; joints [36.914, -37.974, 88.896, -136.238, 60.298, 155.529] to (-279.45, 302.39, -30) mm, rotated rx -180 ry 0 rz 0.01 deg; joints [37.019, -37.873, 88.681, -136.084, 60.262, 155.383]
  MoveC 2806 to (-280.31, 304.94, -30) mm, rotated rx 180 ry 0 rz 0.01 deg; joints [37.072, -37.761, 88.442, -135.979, 60.194, 155.254] to (-282.77, 306.03, -30) mm, rotated rx 180 ry 0 rz 0.01 deg; joints [37.051, -37.626, 88.16, -135.942, 60.078, 155.147]
  MoveL 2807 to (-366.76, 306.02, -30) mm, rotated rx -180 ry 0 rz 0.01 deg; joints [35.369, -33.953, 80.52, -135.993, 56.452, 152.847]
  MoveC 2808 to (-369.48, 304.9, -30) mm, rotated rx 180 ry 0 rz 0.01 deg; joints [35.286, -33.863, 80.334, -136.037, 56.344, 152.816] to (-370.61, 302.17, -30) mm, rotated rx 180 ry 0 rz 0.01 deg; joints [35.19, -33.898, 80.411, -136.157, 56.328, 152.908]
  MoveL 2809 to (-370.6, 98.58, -30) mm, rotated rx -180 ry 0 rz 0.01 deg; joints [29.283, -39.485, 92.377, -145.121, 58.837, 161.197]
  MoveC 2810 to (-369.52, 95.84, -30) mm, rotated rx 180 ry 0 rz 0.01 deg; joints [29.217, -39.595, 92.613, -145.237, 58.917, 161.319] to (-366.86, 94.57, -30) mm, rotated rx 180 ry 0 rz 0.01 deg; joints [29.224, -39.738, 92.916, -145.284, 59.05, 161.422]
  MoveC 2811 to (-360.78, 93.93, -30) mm, rotated rx 180 ry 0 rz 0.01 deg; joints [29.31, -40.012, 93.492, -145.293, 59.328, 161.573] to (-354.75, 92.89, -30) mm, rotated rx 180 ry 0 rz 0.01 deg; joints [29.383, -40.291, 94.08, -145.317, 59.607, 161.736]
  MoveC 2812 to (-348.82, 91.34, -30) mm, rotated rx -180 ry 0 rz 0.01 deg; joints [29.439, -40.575, 94.681, -145.36, 59.886, 161.913] to (-343.08, 89.2, -30) mm, rotated rx -180 ry 0 rz 0.01 deg; joints [29.473, -40.863, 95.291, -145.428, 60.162, 162.105]
  MoveC 2813 to (-326.8, 78.84, -30) mm, rotated rx -180 ry 0 rz 0.01 deg; joints [29.437, -41.764, 97.209, -145.792, 60.99, 162.784] to (-314.52, 63.96, -30) mm, rotated rx -180 ry 0 rz 0.01 deg; joints [29.181, -42.585, 98.971, -146.356, 61.69, 163.518]
  MoveL 2814 to (-295.33, 31.02, -30) mm, rotated rx -180 ry 0 rz 0.01 deg; joints [28.449, -44.032, 102.101, -147.628, 62.886, 164.929]
  MoveC 2815 to (-292.37, 25.07, -30) mm, rotated rx 180 ry 0 rz 0.01 deg; joints [28.304, -44.268, 102.613, -147.86, 63.079, 165.167] to (-290.16, 18.8, -30) mm, rotated rx 180 ry 0 rz 0.01 deg; joints [28.134, -44.478, 103.074, -148.11, 63.244, 165.4]
  MoveC 2816 to (-288.64, 12.34, -30) mm, rotated rx 180 ry 0 rz 0.01 deg; joints [27.944, -44.665, 103.484, -148.373, 63.382, 165.626] to (-287.71, 5.76, -30) mm, rotated rx 180 ry 0 rz 0.01 deg; joints [27.739, -44.829, 103.846, -148.646, 63.496, 165.843]
  MoveC 2817 to (-286.34, 3.02, -30) mm, rotated rx 180 ry 0 rz 0.01 deg; joints [27.67, -44.935, 104.078, -148.752, 63.585, 165.949] to (-283.48, 1.91, -30) mm, rotated rx -180 ry 0 rz 0.01 deg; joints [27.683, -45.067, 104.361, -148.777, 63.718, 166.03]
  MoveL 2818 to (-110.06, 1.91, -30) mm, rotated rx -180 ry 0 rz 0.01 deg; joints [31.124, -51.234, 117.7, -146.761, 70.62, 168.737]
  MoveC 2819 to (-107.15, 3.04, -30) mm, rotated rx -180 ry 0 rz 0.01 deg; joints [31.229, -51.309, 117.861, -146.668, 70.715, 168.75] to (-105.75, 5.83, -30) mm, rotated rx 180 ry 0 rz 0.01 deg; joints [31.362, -51.302, 117.839, -146.528, 70.732, 168.694]
  MoveC 2820 to (-104.81, 12.5, -30) mm, rotated rx 180 ry 0 rz 0.01 deg; joints [31.626, -51.206, 117.613, -146.23, 70.682, 168.525] to (-103.25, 19.05, -30) mm, rotated rx 180 ry 0 rz 0.01 deg; joints [31.898, -51.131, 117.435, -145.929, 70.657, 168.368]
  MoveC 2821 to (-101, 25.39, -30) mm, rotated rx -180 ry 0 rz 0.01 deg; joints [32.178, -51.082, 117.313, -145.626, 70.66, 168.226] to (-97.99, 31.42, -30) mm, rotated rx -180 ry 0 rz 0.01 deg; joints [32.463, -51.062, 117.256, -145.324, 70.695, 168.103]
  MoveC 2822 to (-91.94, 42.13, -30) mm, rotated rx 180 ry 0 rz 0.01 deg; joints [32.985, -51.045, 117.197, -144.778, 70.781, 167.895] to (-86.11, 52.97, -30) mm, rotated rx -180 ry 0 rz 0.01 deg; joints [33.505, -51.015, 117.108, -144.231, 70.855, 167.677]
  MoveC 2823 to (-79.72, 63.51, -30) mm, rotated rx 180 ry 0 rz 0.01 deg; joints [34.028, -51.005, 117.062, -143.686, 70.952, 167.474] to (-72.1, 73.2, -30) mm, rotated rx -180 ry 0 rz 0.01 deg; joints [34.55, -51.047, 117.134, -143.157, 71.102, 167.312]
  MoveC 2824 to (-63.24, 81.44, -30) mm, rotated rx -180 ry 0 rz 0.01 deg; joints [35.052, -51.154, 117.351, -142.665, 71.312, 167.211] to (-53, 87.89, -30) mm, rotated rx 180 ry 0 rz 0.01 deg; joints [35.529, -51.338, 117.743, -142.22, 71.593, 167.184]
  MoveC 2825 to (-41.71, 92.28, -30) mm, rotated rx 180 ry 0 rz 0.01 deg; joints [35.963, -51.595, 118.298, -141.837, 71.935, 167.234] to (-29.79, 94.38, -30) mm, rotated rx -180 ry 0 rz 0.01 deg; joints [36.339, -51.917, 119.001, -141.53, 72.325, 167.361]
  MoveC 2826 to (-29.02, 94.43, -30) mm, rotated rx 180 ry 0 rz 0.01 deg; joints [36.36, -51.939, 119.051, -141.514, 72.352, 167.372] to (-28.25, 94.45, -30) mm, rotated rx 180 ry 0 rz 0.01 deg; joints [36.381, -51.962, 119.102, -141.498, 72.378, 167.383]
  MoveC 2827 to (-27.48, 94.47, -30) mm, rotated rx 180 ry 0 rz 0.01 deg; joints [36.402, -51.985, 119.152, -141.483, 72.405, 167.395] to (-26.71, 94.52, -30) mm, rotated rx 180 ry 0 rz 0.01 deg; joints [36.423, -52.008, 119.202, -141.466, 72.431, 167.406]
  MoveC 2828 to (-24, 95.83, -30) mm, rotated rx 180 ry 0 rz 0.01 deg; joints [36.538, -52.062, 119.318, -141.361, 72.508, 167.41] to (-22.9, 98.63, -30) mm, rotated rx 180 ry 0 rz 0.01 deg; joints [36.664, -52.035, 119.253, -141.226, 72.508, 167.345]
  MoveL 2829 to (-22.91, 302.18, -30) mm, rotated rx 180 ry 0 rz 0.01 deg; joints [43.107, -46.99, 107.936, -133.262, 69.819, 160.668]
  MoveC 2830 to (-24.04, 304.9, -30) mm, rotated rx -180 ry 0 rz 0.01 deg; joints [43.155, -46.879, 107.694, -133.179, 69.746, 160.549] to (-26.76, 306.03, -30) mm, rotated rx 180 ry 0 rz 0.01 deg; joints [43.114, -46.763, 107.444, -133.184, 69.64, 160.46]
  MoveL 2831 to (-110.78, 306.03, -30) mm, rotated rx 180 ry 0 rz 0.01 deg; joints [40.953, -44.047, 101.659, -134.461, 66.715, 158.902]
  MoveC 2832 to (-113.22, 304.94, -30) mm, rotated rx 180 ry 0 rz 0.01 deg; joints [40.862, -43.996, 101.551, -134.535, 66.641, 158.896] to (-114.04, 302.38, -30) mm, rotated rx 180 ry 0 rz 0.01 deg; joints [40.769, -44.041, 101.651, -134.645, 66.644, 158.976]
  MoveC 2833 to (-115.31, 282.54, -30) mm, rotated rx -180 ry 0 rz 0.01 deg; joints [40.168, -44.556, 102.776, -135.437, 66.849, 159.69] to (-123.3, 264.33, -30) mm, rotated rx -180 ry 0 rz 0.01 deg; joints [39.442, -44.786, 103.293, -136.258, 66.79, 160.205]
  MoveC 2834 to (-136.43, 249.55, -30) mm, rotated rx 180 ry 0 rz 0.01 deg; joints [38.69, -44.735, 103.209, -137.012, 66.496, 160.491] to (-153.12, 238.93, -30) mm, rotated rx 180 ry 0 rz 0.01 deg; joints [37.981, -44.44, 102.598, -137.641, 66.012, 160.557]
  MoveC 2835 to (-158.14, 236.98, -30) mm, rotated rx -180 ry 0 rz 0.01 deg; joints [37.806, -44.315, 102.336, -137.779, 65.848, 160.531] to (-163.36, 235.64, -30) mm, rotated rx 180 ry 0 rz 0.01 deg; joints [37.646, -44.167, 102.024, -137.894, 65.669, 160.479]
  MoveC 2836 to (-168.66, 234.7, -30) mm, rotated rx -180 ry 0 rz 0.01 deg; joints [37.496, -44.004, 101.68, -137.993, 65.482, 160.412] to (-173.99, 233.94, -30) mm, rotated rx 180 ry 0 rz 0.01 deg; joints [37.351, -43.834, 101.322, -138.084, 65.289, 160.336]
  MoveL 2837 to (-214.9, 233.65, -30) mm, rotated rx 180 ry 0 rz 0.01 deg; joints [36.431, -42.349, 98.181, -138.508, 63.717, 159.534]
  MoveC 2838 to (-240.66, 238.89, -30) mm, rotated rx 180 ry 0 rz 0.01 deg; joints [36.029, -41.233, 95.819, -138.507, 62.632, 158.802] to (-262.34, 253.78, -30) mm, rotated rx -180 ry 0 rz 0.01 deg; joints [36.004, -39.977, 93.157, -138.038, 61.573, 157.756]
  MoveC 2839 to (-274.89, 272.82, -30) mm, rotated rx 180 ry 0 rz 0.01 deg; joints [36.286, -38.933, 90.941, -137.31, 60.822, 156.71] to (-279.69, 295.12, -30) mm, rotated rx 180 ry 0 rz 0.01 deg; joints [36.813, -38.082, 89.128, -136.392, 60.344, 155.681]
  MoveC 2840 to (-278.46, 299.32, -30) mm, rotated rx 180 ry 0 rz 0.01 deg; joints [36.955, -38.007, 88.964, -136.21, 60.342, 155.536] to (-275.01, 302.01, -30) mm, rotated rx 180 ry 0 rz 0.01 deg; joints [37.102, -38.067, 89.086, -136.082, 60.45, 155.508]
  MoveC 2841 to (-271.47, 304.45, -30) mm, rotated rx -180 ry 0 rz 0.01 deg; joints [37.244, -38.137, 89.23, -135.964, 60.565, 155.493] to (-269.57, 308.31, -30) mm, rotated rx 180 ry 0 rz 0.01 deg; joints [37.391, -38.098, 89.141, -135.793, 60.594, 155.378]
  MoveC 2842 to (-269.28, 309.83, -30) mm, rotated rx 180 ry 0 rz 0.01 deg; joints [37.439, -38.063, 89.067, -135.728, 60.587, 155.321] to (-269.02, 311.37, -30) mm, rotated rx 180 ry 0 rz 0.01 deg; joints [37.487, -38.027, 88.989, -135.662, 60.578, 155.263]
  MoveC 2843 to (-269.76, 313.93, -30) mm, rotated rx 180 ry 0 rz 0.01 deg; joints [37.542, -37.919, 88.76, -135.557, 60.515, 155.137] to (-272.18, 315.04, -30) mm, rotated rx -180 ry 0 rz 0.01 deg; joints [37.521, -37.786, 88.48, -135.521, 60.402, 155.03]
  MoveL 2844 to (-375.78, 315.04, -30) mm, rotated rx -180 ry 0 rz 0.01 deg; joints [35.439, -33.237, 79.023, -135.554, 55.926, 152.149]
  MoveC 2845 to (-378.5, 313.91, -30) mm, rotated rx 180 ry 0 rz 0.01 deg; joints [35.357, -33.145, 78.834, -135.595, 55.817, 152.117] to (-379.63, 311.19, -30) mm, rotated rx -180 ry 0 rz 0.01 deg; joints [35.262, -33.181, 78.913, -135.715, 55.801, 152.21]
  MoveL 2846 to (-379.62, 88.72, -30) mm, rotated rx 180 ry 0 rz 0.01 deg; joints [28.823, -39.323, 92.056, -145.572, 58.547, 161.359]
  MoveC 2847 to (-378.55, 86.29, -30) mm, rotated rx 180 ry 0 rz 0.01 deg; joints [28.766, -39.426, 92.275, -145.675, 58.623, 161.469] to (-376.03, 85.45, -30) mm, rotated rx -180 ry 0 rz 0.01 deg; joints [28.783, -39.554, 92.545, -145.705, 58.746, 161.553]
  MoveC 2848 to (-355.28, 83.75, -30) mm, rotated rx 180 ry 0 rz 0.01 deg; joints [29.088, -40.476, 94.486, -145.712, 59.69, 162.046] to (-336.39, 74.99, -30) mm, rotated rx -180 ry 0 rz 0.01 deg; joints [29.143, -41.457, 96.567, -146.006, 60.619, 162.728]
  MoveC 2849 to (-332.59, 71.93, -30) mm, rotated rx -180 ry 0 rz 0.01 deg; joints [29.113, -41.68, 97.044, -146.118, 60.82, 162.906] to (-329.2, 68.42, -30) mm, rotated rx -180 ry 0 rz 0.01 deg; joints [29.061, -41.895, 97.504, -146.25, 61.007, 163.091]
  MoveC 2850 to (-326.1, 64.65, -30) mm, rotated rx 180 ry 0 rz 0.01 deg; joints [28.996, -42.103, 97.95, -146.394, 61.185, 163.276] to (-323.13, 60.79, -30) mm, rotated rx 180 ry 0 rz 0.01 deg; joints [28.925, -42.306, 98.387, -146.542, 61.358, 163.461]
  MoveL 2851 to (-303.14, 26.52, -30) mm, rotated rx -180 ry 0 rz 0.01 deg; joints [28.16, -43.816, 101.651, -147.876, 62.606, 164.935]
  MoveC 2852 to (-300.35, 20.8, -30) mm, rotated rx -180 ry 0 rz 0.01 deg; joints [28.019, -44.041, 102.139, -148.099, 62.79, 165.163] to (-298.36, 14.77, -30) mm, rotated rx 180 ry 0 rz 0.01 deg; joints [27.853, -44.238, 102.571, -148.342, 62.943, 165.385]
  MoveC 2853 to (-297.06, 8.55, -30) mm, rotated rx 180 ry 0 rz 0.01 deg; joints [27.667, -44.411, 102.951, -148.598, 63.069, 165.6] to (-296.31, 2.25, -30) mm, rotated rx 180 ry 0 rz 0.01 deg; joints [27.468, -44.563, 103.287, -148.861, 63.172, 165.806]
  MoveC 2854 to (-296.26, 0.83, -30) mm, rotated rx 180 ry 0 rz 0.01 deg; joints [27.421, -44.592, 103.351, -148.921, 63.19, 165.85] to (-296.34, -0.58, -30) mm, rotated rx -180 ry 0 rz 0.01 deg; joints [27.372, -44.616, 103.406, -148.982, 63.203, 165.892]
  MoveC 2855 to (-296.46, -2, -30) mm, rotated rx 180 ry 0 rz 0.01 deg; joints [27.322, -44.639, 103.457, -149.043, 63.214, 165.933] to (-296.54, -3.41, -30) mm, rotated rx 180 ry 0 rz 0.01 deg; joints [27.272, -44.663, 103.51, -149.104, 63.226, 165.975]
  MoveC 2856 to (-295.57, -6.01, -30) mm, rotated rx 180 ry 0 rz 0.01 deg; joints [27.201, -44.75, 103.702, -149.208, 63.297, 166.07] to (-293.01, -7.11, -30) mm, rotated rx -180 ry 0 rz 0.01 deg; joints [27.209, -44.871, 103.961, -149.236, 63.418, 166.146]
  MoveL 2857 to (-100.5, -7.11, -30) mm, rotated rx -180 ry 0 rz 0.01 deg; joints [31.004, -51.715, 118.778, -146.998, 71.094, 169.124]
  MoveC 2858 to (-97.94, -6.01, -30) mm, rotated rx 180 ry 0 rz 0.01 deg; joints [31.101, -51.778, 118.914, -146.911, 71.176, 169.133] to (-96.97, -3.41, -30) mm, rotated rx 180 ry 0 rz 0.01 deg; joints [31.219, -51.761, 118.871, -146.784, 71.18, 169.077]
  MoveC 2859 to (-97.08, 1.12, -30) mm, rotated rx 180 ry 0 rz 0.01 deg; joints [31.383, -51.673, 118.666, -146.593, 71.117, 168.953] to (-97.01, 5.65, -30) mm, rotated rx -180 ry 0 rz 0.01 deg; joints [31.551, -51.59, 118.473, -146.399, 71.062, 168.831]
  MoveC 2860 to (-96.5, 10.17, -30) mm, rotated rx 180 ry 0 rz 0.01 deg; joints [31.728, -51.521, 118.311, -146.199, 71.023, 168.715] to (-95.32, 14.56, -30) mm, rotated rx -180 ry 0 rz 0.01 deg; joints [31.914, -51.475, 118.202, -145.994, 71.011, 168.613]
  MoveC 2861 to (-94.2, 17.71, -30) mm, rotated rx 180 ry 0 rz 0.01 deg; joints [32.054, -51.451, 118.142, -145.843, 71.012, 168.543] to (-93.04, 20.85, -30) mm, rotated rx 180 ry 0 rz 0.01 deg; joints [32.195, -51.428, 118.084, -145.692, 71.015, 168.474]
  MoveC 2862 to (-91.73, 23.94, -30) mm, rotated rx 180 ry 0 rz 0.01 deg; joints [32.336, -51.411, 118.038, -145.54, 71.023, 168.408] to (-90.18, 26.91, -30) mm, rotated rx 180 ry 0 rz 0.01 deg; joints [32.479, -51.403, 118.015, -145.39, 71.043, 168.349]
  MoveL 2863 to (-69.87, 61.52, -30) mm, rotated rx 180 ry 0 rz 0.01 deg; joints [34.193, -51.36, 117.845, -143.604, 71.336, 167.685]
  MoveC 2864 to (-62.89, 69.4, -30) mm, rotated rx 180 ry 0 rz 0.01 deg; joints [34.639, -51.417, 117.955, -143.157, 71.484, 167.567] to (-54.99, 76.34, -30) mm, rotated rx -180 ry 0 rz 0.01 deg; joints [35.077, -51.521, 118.167, -142.731, 71.675, 167.49]
  MoveC 2865 to (-45.89, 81.75, -30) mm, rotated rx 180 ry 0 rz 0.01 deg; joints [35.491, -51.69, 118.529, -142.345, 71.927, 167.476] to (-35.77, 84.81, -30) mm, rotated rx -180 ry 0 rz 0.01 deg; joints [35.853, -51.938, 119.068, -142.034, 72.244, 167.547]
  MoveC 2866 to (-31.22, 85.44, -30) mm, rotated rx 180 ry 0 rz 0.01 deg; joints [35.99, -52.064, 119.345, -141.924, 72.396, 167.6] to (-26.65, 85.74, -30) mm, rotated rx 180 ry 0 rz 0.01 deg; joints [36.118, -52.197, 119.638, -141.825, 72.552, 167.663]
  MoveC 2867 to (-22.06, 85.74, -30) mm, rotated rx 180 ry 0 rz 0.01 deg; joints [36.236, -52.337, 119.946, -141.738, 72.712, 167.735] to (-17.48, 85.45, -30) mm, rotated rx 180 ry 0 rz 0.01 deg; joints [36.344, -52.482, 120.267, -141.662, 72.876, 167.816]
  MoveC 2868 to (-14.96, 86.29, -30) mm, rotated rx -180 ry 0 rz 0.01 deg; joints [36.438, -52.54, 120.394, -141.579, 72.952, 167.831] to (-13.89, 88.72, -30) mm, rotated rx -180 ry 0 rz 0.01 deg; joints [36.552, -52.521, 120.346, -141.458, 72.956, 167.777]
  MoveL 2869 to (-13.89, 311.2, -30) mm, rotated rx 180 ry 0 rz 0.01 deg; joints [43.609, -47.012, 107.97, -132.766, 70.005, 160.5]
  MoveC 2870 to (-15.02, 313.92, -30) mm, rotated rx -180 ry 0 rz 0.01 deg; joints [43.656, -46.9, 107.726, -132.684, 69.932, 160.381] to (-17.75, 315.05, -30) mm, rotated rx 180 ry 0 rz 0.01 deg; joints [43.614, -46.785, 107.477, -132.689, 69.827, 160.291]
  MoveL 2871 to (-121.33, 315.05, -30) mm, rotated rx -180 ry 0 rz 0.01 deg; joints [40.949, -43.428, 100.335, -134.245, 66.22, 158.353]
  MoveC 2872 to (-123.73, 313.95, -30) mm, rotated rx -180 ry 0 rz 0.01 deg; joints [40.859, -43.378, 100.229, -134.318, 66.147, 158.348] to (-124.47, 311.41, -30) mm, rotated rx 180 ry 0 rz 0.01 deg; joints [40.77, -43.426, 100.335, -134.426, 66.152, 158.43]
  MoveC 2873 to (-123.68, 306.37, -30) mm, rotated rx -180 ry 0 rz 0.01 deg; joints [40.646, -43.598, 100.707, -134.613, 66.244, 158.637] to (-122.81, 301.34, -30) mm, rotated rx 180 ry 0 rz 0.01 deg; joints [40.525, -43.772, 101.082, -134.799, 66.34, 158.845]
  MoveC 2874 to (-122.42, 296.23, -30) mm, rotated rx -180 ry 0 rz 0.01 deg; joints [40.388, -43.931, 101.427, -134.994, 66.418, 159.045] to (-123.08, 291.14, -30) mm, rotated rx 180 ry 0 rz 0.01 deg; joints [40.226, -44.051, 101.691, -135.202, 66.459, 159.222]
  MoveC 2875 to (-125.14, 283.59, -30) mm, rotated rx 180 ry 0 rz 0.01 deg; joints [39.959, -44.193, 102.002, -135.524, 66.479, 159.463] to (-127.71, 276.2, -30) mm, rotated rx 180 ry 0 rz 0.01 deg; joints [39.682, -44.31, 102.262, -135.847, 66.479, 159.687]
  MoveC 2876 to (-131.15, 269.15, -30) mm, rotated rx -180 ry 0 rz 0.01 deg; joints [39.394, -44.386, 102.436, -136.169, 66.442, 159.88] to (-135.73, 262.77, -30) mm, rotated rx 180 ry 0 rz 0.01 deg; joints [39.098, -44.403, 102.481, -136.479, 66.355, 160.026]
  MoveC 2877 to (-143.17, 255.52, -30) mm, rotated rx -180 ry 0 rz 0.01 deg; joints [38.707, -44.342, 102.363, -136.859, 66.172, 160.147] to (-151.79, 249.72, -30) mm, rotated rx -180 ry 0 rz 0.01 deg; joints [38.333, -44.198, 102.067, -137.195, 65.925, 160.193]
  MoveC 2878 to (-161.34, 245.6, -30) mm, rotated rx -180 ry 0 rz 0.01 deg; joints [37.989, -43.973, 101.597, -137.472, 65.62, 160.158] to (-171.48, 243.34, -30) mm, rotated rx -180 ry 0 rz 0.01 deg; joints [37.688, -43.674, 100.966, -137.678, 65.266, 160.044]
  MoveL 2879 to (-214.9, 242.66, -30) mm, rotated rx 180 ry 0 rz 0.01 deg; joints [36.696, -42.107, 97.655, -138.139, 63.604, 159.199]
  MoveC 2880 to (-228.71, 244.47, -30) mm, rotated rx -180 ry 0 rz 0.01 deg; joints [36.449, -41.537, 96.451, -138.183, 63.038, 158.843] to (-241.58, 249.79, -30) mm, rotated rx -180 ry 0 rz 0.01 deg; joints [36.327, -40.899, 95.099, -138.064, 62.46, 158.367]
  MoveC 2881 to (-252.8, 257.98, -30) mm, rotated rx 180 ry 0 rz 0.01 deg; joints [36.326, -40.235, 93.691, -137.802, 61.907, 157.804] to (-261.98, 268.41, -30) mm, rotated rx -180 ry 0 rz 0.01 deg; joints [36.431, -39.577, 92.297, -137.425, 61.405, 157.186]
  MoveC 2882 to (-269.32, 284.15, -30) mm, rotated rx 180 ry 0 rz 0.01 deg; joints [36.722, -38.828, 90.704, -136.807, 60.908, 156.382] to (-270.8, 301.46, -30) mm, rotated rx 180 ry 0 rz 0.01 deg; joints [37.175, -38.255, 89.48, -136.087, 60.63, 155.634]
  MoveC 2883 to (-270.49, 303.96, -30) mm, rotated rx 180 ry 0 rz 0.01 deg; joints [37.251, -38.192, 89.345, -135.98, 60.611, 155.537] to (-269.99, 306.43, -30) mm, rotated rx 180 ry 0 rz 0.01 deg; joints [37.33, -38.138, 89.228, -135.874, 60.6, 155.446]
  MoveC 2884 to (-269.78, 307.37, -30) mm, rotated rx 180 ry 0 rz 0.01 deg; joints [37.36, -38.118, 89.185, -135.834, 60.598, 155.412] to (-269.57, 308.31, -30) mm, rotated rx 180 ry 0 rz 0.01 deg; joints [37.391, -38.098, 89.141, -135.793, 60.594, 155.378]
  MoveC 2885 to (-267.64, 311.81, -30) mm, rotated rx -180 ry 0 rz 0.01 deg; joints [37.528, -38.07, 89.078, -135.637, 60.629, 155.278] to (-264.05, 313.6, -30) mm, rotated rx -180 ry 0 rz 0.01 deg; joints [37.654, -38.161, 89.265, -135.546, 60.753, 155.291]
  MoveC 2886 to (-260.43, 315.15, -30) mm, rotated rx -180 ry 0 rz 0.01 deg; joints [37.773, -38.26, 89.47, -135.464, 60.881, 155.315] to (-257.94, 318.2, -30) mm, rotated rx -180 ry 0 rz 0.01 deg; joints [37.911, -38.267, 89.48, -135.324, 60.944, 155.247]
  MoveC 2887 to (-257.41, 319.29, -30) mm, rotated rx -180 ry 0 rz 0.01 deg; joints [37.952, -38.255, 89.454, -135.276, 60.951, 155.214] to (-256.85, 320.36, -30) mm, rotated rx 180 ry 0 rz 0.01 deg; joints [37.993, -38.245, 89.431, -135.229, 60.961, 155.183]
  MoveC 2888 to (-256.89, 322.62, -30) mm, rotated rx 180 ry 0 rz 0.01 deg; joints [38.054, -38.173, 89.278, -135.135, 60.93, 155.086] to (-258.86, 323.74, -30) mm, rotated rx 180 ry 0 rz 0.01 deg; joints [38.043, -38.06, 89.039, -135.097, 60.836, 154.991]
  MoveL 2889 to (-384.47, 323.74, -30) mm, rotated rx 180 ry 0 rz 0.01 deg; joints [35.506, -32.533, 77.552, -135.116, 55.414, 151.456]
  MoveC 2890 to (-387.19, 322.61, -30) mm, rotated rx -180 ry 0 rz 0.01 deg; joints [35.424, -32.439, 77.36, -135.154, 55.304, 151.422] to (-388.32, 319.88, -30) mm, rotated rx -180 ry 0 rz 0.01 deg; joints [35.33, -32.476, 77.441, -135.275, 55.288, 151.517]
  MoveL 2891 to (-388.32, 77.01, -30) mm, rotated rx -180 ry 0 rz 0.01 deg; joints [28.312, -39.213, 91.844, -146.1, 58.289, 161.593]
  MoveC 2892 to (-387.19, 74.77, -30) mm, rotated rx -180 ry 0 rz 0.01 deg; joints [28.261, -39.312, 92.057, -146.195, 58.366, 161.697] to (-384.73, 74.34, -30) mm, rotated rx -180 ry 0 rz 0.01 deg; joints [28.289, -39.429, 92.303, -146.209, 58.482, 161.765]
  MoveC 2893 to (-382.02, 75.2, -30) mm, rotated rx -180 ry 0 rz 0.01 deg; joints [28.361, -39.527, 92.507, -146.165, 58.595, 161.792] to (-379.34, 76.16, -30) mm, rotated rx 180 ry 0 rz 0.01 deg; joints [28.437, -39.621, 92.703, -146.117, 58.705, 161.814]
  MoveC 2894 to (-376.6, 76.94, -30) mm, rotated rx -180 ry 0 rz 0.01 deg; joints [28.507, -39.722, 92.914, -146.076, 58.82, 161.844] to (-373.76, 77.23, -30) mm, rotated rx 180 ry 0 rz 0.01 deg; joints [28.565, -39.838, 93.156, -146.055, 58.944, 161.893]
  MoveC 2895 to (-364.53, 76.76, -30) mm, rotated rx 180 ry 0 rz 0.01 deg; joints [28.708, -40.242, 94.006, -146.047, 59.361, 162.101] to (-355.46, 75.06, -30) mm, rotated rx -180 ry 0 rz 0.01 deg; joints [28.811, -40.663, 94.895, -146.087, 59.783, 162.346]
  MoveC 2896 to (-346.83, 71.63, -30) mm, rotated rx -180 ry 0 rz 0.01 deg; joints [28.853, -41.099, 95.82, -146.199, 60.203, 162.637] to (-339.31, 66.18, -30) mm, rotated rx 180 ry 0 rz 0.01 deg; joints [28.811, -41.53, 96.737, -146.397, 60.594, 162.97]
  MoveC 2897 to (-336.38, 63.31, -30) mm, rotated rx -180 ry 0 rz 0.01 deg; joints [28.771, -41.712, 97.127, -146.506, 60.755, 163.124] to (-333.6, 60.31, -30) mm, rotated rx -180 ry 0 rz 0.01 deg; joints [28.724, -41.891, 97.51, -146.62, 60.91, 163.279]
  MoveC 2898 to (-331.04, 57.1, -30) mm, rotated rx -180 ry 0 rz 0.01 deg; joints [28.666, -42.064, 97.882, -146.744, 61.058, 163.434] to (-328.81, 53.66, -30) mm, rotated rx -180 ry 0 rz 0.01 deg; joints [28.594, -42.228, 98.235, -146.879, 61.194, 163.591]
  MoveL 2899 to (-308.02, 16.23, -30) mm, rotated rx -180 ry 0 rz 0.01 deg; joints [27.732, -43.83, 101.699, -148.348, 62.515, 165.173]
  MoveC 2900 to (-305.83, 9.29, -30) mm, rotated rx 180 ry 0 rz 0.01 deg; joints [27.538, -44.053, 102.187, -148.629, 62.687, 165.427] to (-304.94, 2.07, -30) mm, rotated rx -180 ry 0 rz 0.01 deg; joints [27.311, -44.229, 102.575, -148.931, 62.807, 165.666]
  MoveC 2901 to (-305.17, -5.18, -30) mm, rotated rx 180 ry 0 rz 0.01 deg; joints [27.063, -44.359, 102.867, -149.243, 62.879, 165.885] to (-306.32, -12.35, -30) mm, rotated rx 180 ry 0 rz 0.01 deg; joints [26.8, -44.45, 103.075, -149.557, 62.91, 166.084]
  MoveC 2902 to (-305.77, -14.74, -30) mm, rotated rx 180 ry 0 rz 0.01 deg; joints [26.728, -44.517, 103.221, -149.656, 62.96, 166.165] to (-303.57, -15.8, -30) mm, rotated rx -180 ry 0 rz 0.01 deg; joints [26.73, -44.623, 103.45, -149.685, 63.066, 166.234]
  MoveL 2903 to (-89.95, -15.8, -30) mm, rotated rx 180 ry 0 rz 0.01 deg; joints [30.916, -52.217, 119.905, -147.203, 71.601, 169.513]
  MoveC 2904 to (-87.74, -14.74, -30) mm, rotated rx -180 ry 0 rz 0.01 deg; joints [31.005, -52.268, 120.017, -147.122, 71.67, 169.517] to (-87.19, -12.35, -30) mm, rotated rx 180 ry 0 rz 0.01 deg; joints [31.107, -52.242, 119.954, -147.011, 71.66, 169.462]
  MoveC 2905 to (-88.17, -6.99, -30) mm, rotated rx -180 ry 0 rz 0.01 deg; joints [31.284, -52.112, 119.654, -146.797, 71.555, 169.305] to (-88.67, -1.57, -30) mm, rotated rx -180 ry 0 rz 0.01 deg; joints [31.474, -51.995, 119.384, -146.573, 71.466, 169.152]
  MoveC 2906 to (-88.58, 3.88, -30) mm, rotated rx -180 ry 0 rz 0.01 deg; joints [31.677, -51.896, 119.152, -146.34, 71.399, 169.006] to (-87.79, 9.28, -30) mm, rotated rx 180 ry 0 rz 0.01 deg; joints [31.893, -51.819, 118.971, -146.097, 71.359, 168.871]
  MoveC 2907 to (-87, 12.3, -30) mm, rotated rx 180 ry 0 rz 0.01 deg; joints [32.021, -51.787, 118.894, -145.956, 71.349, 168.8] to (-85.92, 15.23, -30) mm, rotated rx -180 ry 0 rz 0.01 deg; joints [32.153, -51.766, 118.84, -145.815, 71.351, 168.737]
  MoveL 2908 to (-83.71, 20.43, -30) mm, rotated rx -180 ry 0 rz 0.01 deg; joints [32.393, -51.737, 118.764, -145.558, 71.366, 168.627]
  MoveL 2909 to (-64.5, 53.96, -30) mm, rotated rx 180 ry 0 rz 0.01 deg; joints [34.054, -51.684, 118.574, -143.827, 71.629, 167.984]
  MoveC 2910 to (-57.17, 63.43, -30) mm, rotated rx 180 ry 0 rz 0.01 deg; joints [34.568, -51.721, 118.635, -143.305, 71.769, 167.829] to (-47.57, 70.59, -30) mm, rotated rx -180 ry 0 rz 0.01 deg; joints [35.058, -51.872, 118.953, -142.837, 72.017, 167.773]
  MoveC 2911 to (-36.57, 75.23, -30) mm, rotated rx -180 ry 0 rz 0.01 deg; joints [35.496, -52.115, 119.48, -142.444, 72.345, 167.812] to (-24.83, 77.41, -30) mm, rotated rx -180 ry 0 rz 0.01 deg; joints [35.871, -52.429, 120.167, -142.134, 72.728, 167.933]
  MoveC 2912 to (-20.71, 77.37, -30) mm, rotated rx 180 ry 0 rz 0.01 deg; joints [35.975, -52.555, 120.446, -142.057, 72.873, 167.999] to (-16.66, 76.61, -30) mm, rotated rx -180 ry 0 rz 0.01 deg; joints [36.052, -52.693, 120.754, -142.01, 73.025, 168.084]
  MoveC 2913 to (-12.71, 75.48, -30) mm, rotated rx -180 ry 0 rz 0.01 deg; joints [36.114, -52.836, 121.072, -141.98, 73.177, 168.178] to (-8.77, 74.31, -30) mm, rotated rx 180 ry 0 rz 0.01 deg; joints [36.175, -52.978, 121.391, -141.951, 73.33, 168.273]
  MoveC 2914 to (-6.31, 74.74, -30) mm, rotated rx 180 ry 0 rz 0.01 deg; joints [36.255, -53.043, 121.534, -141.885, 73.409, 168.299] to (-5.19, 76.97, -30) mm, rotated rx 180 ry 0 rz 0.01 deg; joints [36.363, -53.03, 121.5, -141.77, 73.418, 168.253]
  MoveL 2915 to (-5.2, 319.89, -30) mm, rotated rx -180 ry 0 rz 0.01 deg; joints [44.094, -47.029, 107.992, -132.286, 70.182, 160.336]
  MoveC 2916 to (-6.33, 322.62, -30) mm, rotated rx -180 ry 0 rz 0.01 deg; joints [44.14, -46.917, 107.748, -132.205, 70.11, 160.216] to (-9.05, 323.74, -30) mm, rotated rx 180 ry 0 rz 0.01 deg; joints [44.097, -46.802, 107.5, -132.212, 70.005, 160.126]
  MoveL 2917 to (-134.64, 323.74, -30) mm, rotated rx 180 ry 0 rz 0.01 deg; joints [40.87, -42.715, 98.813, -134.066, 65.626, 157.751]
  MoveC 2918 to (-136.61, 322.62, -30) mm, rotated rx 180 ry 0 rz 0.01 deg; joints [40.791, -42.679, 98.739, -134.133, 65.568, 157.755] to (-136.66, 320.36, -30) mm, rotated rx 180 ry 0 rz 0.01 deg; joints [40.726, -42.743, 98.878, -134.222, 65.594, 157.842]
  MoveC 2919 to (-134.15, 314.94, -30) mm, rotated rx 180 ry 0 rz 0.01 deg; joints [40.635, -42.989, 99.406, -134.405, 65.755, 158.102] to (-132.27, 309.27, -30) mm, rotated rx -180 ry 0 rz 0.01 deg; joints [40.52, -43.218, 99.899, -134.605, 65.895, 158.357]
  MoveC 2920 to (-131.18, 303.39, -30) mm, rotated rx -180 ry 0 rz 0.01 deg; joints [40.38, -43.425, 100.346, -134.823, 66.009, 158.602] to (-131.01, 297.41, -30) mm, rotated rx 180 ry 0 rz 0.01 deg; joints [40.214, -43.602, 100.729, -135.055, 66.091, 158.832]
  MoveC 2921 to (-133.65, 283.53, -30) mm, rotated rx 180 ry 0 rz 0.01 deg; joints [39.752, -43.902, 101.386, -135.634, 66.169, 159.301] to (-140.04, 270.92, -30) mm, rotated rx 180 ry 0 rz 0.01 deg; joints [39.233, -44.031, 101.678, -136.21, 66.093, 159.644]
  MoveC 2922 to (-149.91, 260.75, -30) mm, rotated rx 180 ry 0 rz 0.01 deg; joints [38.702, -43.965, 101.556, -136.733, 65.856, 159.827] to (-162.51, 254.25, -30) mm, rotated rx 180 ry 0 rz 0.01 deg; joints [38.217, -43.699, 101.001, -137.14, 65.467, 159.82]
  MoveC 2923 to (-166.45, 253.09, -30) mm, rotated rx 180 ry 0 rz 0.01 deg; joints [38.092, -43.59, 100.774, -137.23, 65.334, 159.786] to (-170.45, 252.17, -30) mm, rotated rx 180 ry 0 rz 0.01 deg; joints [37.973, -43.473, 100.526, -137.312, 65.195, 159.741]
  MoveC 2924 to (-174.51, 251.56, -30) mm, rotated rx -180 ry 0 rz 0.01 deg; joints [37.862, -43.344, 100.254, -137.381, 65.048, 159.683] to (-178.62, 251.36, -30) mm, rotated rx -180 ry 0 rz 0.01 deg; joints [37.762, -43.202, 99.955, -137.433, 64.895, 159.609]
  MoveL 2925 to (-220.94, 251.97, -30) mm, rotated rx 180 ry 0 rz 0.01 deg; joints [36.836, -41.626, 96.627, -137.812, 63.251, 158.723]
  MoveC 2926 to (-241.94, 259.96, -30) mm, rotated rx -180 ry 0 rz 0.01 deg; joints [36.614, -40.602, 94.46, -137.646, 62.319, 157.967] to (-256.92, 276.7, -30) mm, rotated rx 180 ry 0 rz 0.01 deg; joints [36.773, -39.54, 92.206, -137.05, 61.506, 156.972]
  MoveC 2927 to (-262.37, 297.33, -30) mm, rotated rx -180 ry 0 rz 0.01 deg; joints [37.238, -38.719, 90.456, -136.22, 61.027, 156.008] to (-257.94, 318.2, -30) mm, rotated rx 180 ry 0 rz 0.01 deg; joints [37.911, -38.267, 89.48, -135.324, 60.944, 155.247]
  MoveC 2928 to (-255.53, 320.81, -30) mm, rotated rx 180 ry 0 rz 0.01 deg; joints [38.034, -38.284, 89.512, -135.204, 61.009, 155.196] to (-252.05, 321.56, -30) mm, rotated rx 180 ry 0 rz 0.01 deg; joints [38.129, -38.4, 89.753, -135.155, 61.139, 155.249]
  MoveC 2929 to (-248.6, 322.12, -30) mm, rotated rx 180 ry 0 rz 0.01 deg; joints [38.219, -38.52, 90.004, -135.113, 61.272, 155.309] to (-245.85, 324.29, -30) mm, rotated rx -180 ry 0 rz 0.01 deg; joints [38.338, -38.563, 90.091, -135.008, 61.355, 155.284]
  MoveC 2930 to (-244.17, 326.44, -30) mm, rotated rx 180 ry 0 rz 0.01 deg; joints [38.434, -38.564, 90.089, -134.91, 61.395, 155.234] to (-242.42, 328.54, -30) mm, rotated rx 180 ry 0 rz 0.01 deg; joints [38.529, -38.569, 90.096, -134.813, 61.439, 155.188]
  MoveL 2931 to (-242.27, 328.7, -30) mm, rotated rx 180 ry 0 rz 0.01 deg; joints [38.537, -38.57, 90.098, -134.805, 61.443, 155.185]
  MoveL 2932 to (-242.11, 328.87, -30) mm, rotated rx 180 ry 0 rz 0.01 deg; joints [38.545, -38.571, 90.1, -134.798, 61.447, 155.182]
  MoveC 2933 to (-241.78, 330.79, -30) mm, rotated rx -180 ry 0 rz 0.01 deg; joints [38.605, -38.524, 90, -134.716, 61.436, 155.109] to (-243.42, 331.86, -30) mm, rotated rx 180 ry 0 rz 0.01 deg; joints [38.598, -38.427, 89.794, -134.68, 61.357, 155.025]
  MoveL 2934 to (-392.59, 331.86, -30) mm, rotated rx 180 ry 0 rz 0.01 deg; joints [35.568, -31.861, 76.152, -134.692, 54.931, 150.79]
  MoveC 2935 to (-395.31, 330.73, -30) mm, rotated rx -180 ry 0 rz 0.01 deg; joints [35.486, -31.766, 75.957, -134.728, 54.819, 150.753] to (-396.44, 328, -30) mm, rotated rx 180 ry 0 rz 0.01 deg; joints [35.393, -31.804, 76.039, -134.848, 54.803, 150.85]
  MoveL 2936 to (-396.44, 62.49, -30) mm, rotated rx 180 ry 0 rz 0.01 deg; joints [27.725, -39.183, 91.807, -146.749, 58.085, 161.937]
  MoveC 2937 to (-395.32, 60.72, -30) mm, rotated rx 180 ry 0 rz 0.01 deg; joints [27.687, -39.271, 91.995, -146.824, 58.157, 162.024] to (-393.24, 60.95, -30) mm, rotated rx -180 ry 0 rz 0.01 deg; joints [27.729, -39.357, 92.175, -146.81, 58.249, 162.06]
  MoveC 2938 to (-391.49, 62.35, -30) mm, rotated rx -180 ry 0 rz 0.01 deg; joints [27.802, -39.403, 92.268, -146.746, 58.313, 162.047] to (-389.74, 63.75, -30) mm, rotated rx 180 ry 0 rz 0.01 deg; joints [27.875, -39.448, 92.36, -146.681, 58.377, 162.034]
  MoveC 2939 to (-387.85, 64.99, -30) mm, rotated rx 180 ry 0 rz 0.01 deg; joints [27.945, -39.502, 92.473, -146.623, 58.448, 162.03] to (-385.76, 65.85, -30) mm, rotated rx -180 ry 0 rz 0.01 deg; joints [28.006, -39.574, 92.622, -146.581, 58.533, 162.044]
  MoveC 2940 to (-380.35, 67.35, -30) mm, rotated rx -180 ry 0 rz 0.01 deg; joints [28.144, -39.775, 93.04, -146.502, 58.761, 162.104] to (-374.89, 68.66, -30) mm, rotated rx 180 ry 0 rz 0.01 deg; joints [28.277, -39.98, 93.47, -146.43, 58.991, 162.171]
  MoveC 2941 to (-369.29, 69.31, -30) mm, rotated rx -180 ry 0 rz 0.01 deg; joints [28.393, -40.205, 93.942, -146.384, 59.235, 162.264] to (-363.66, 68.81, -30) mm, rotated rx -180 ry 0 rz 0.01 deg; joints [28.473, -40.455, 94.469, -146.387, 59.491, 162.396]
  MoveC 2942 to (-356.43, 66.73, -30) mm, rotated rx 180 ry 0 rz 0.01 deg; joints [28.531, -40.806, 95.211, -146.45, 59.836, 162.614] to (-349.67, 63.41, -30) mm, rotated rx -180 ry 0 rz 0.01 deg; joints [28.543, -41.161, 95.964, -146.564, 60.172, 162.862]
  MoveC 2943 to (-343.62, 58.91, -30) mm, rotated rx 180 ry 0 rz 0.01 deg; joints [28.504, -41.509, 96.707, -146.73, 60.489, 163.132] to (-338.55, 53.34, -30) mm, rotated rx -180 ry 0 rz 0.01 deg; joints [28.413, -41.837, 97.41, -146.944, 60.775, 163.417]
  MoveL 2944 to (-317.71, 18.12, -30) mm, rotated rx 180 ry 0 rz 0.01 deg; joints [27.625, -43.407, 100.798, -148.331, 62.078, 164.944]
  MoveC 2945 to (-314.86, 11.63, -30) mm, rotated rx 180 ry 0 rz 0.01 deg; joints [27.459, -43.65, 101.325, -148.59, 62.274, 165.198] to (-313.48, 4.67, -30) mm, rotated rx 180 ry 0 rz 0.01 deg; joints [27.251, -43.841, 101.745, -148.879, 62.412, 165.44]
  MoveC 2946 to (-313.22, -2.39, -30) mm, rotated rx 180 ry 0 rz 0.01 deg; joints [27.018, -43.988, 102.071, -149.179, 62.502, 165.663] to (-313.67, -9.43, -30) mm, rotated rx -180 ry 0 rz 0.01 deg; joints [26.773, -44.105, 102.334, -149.483, 62.562, 165.872]
  MoveC 2947 to (-314.27, -12.42, -30) mm, rotated rx -180 ry 0 rz 0.01 deg; joints [26.662, -44.138, 102.41, -149.615, 62.569, 165.953] to (-315.39, -15.26, -30) mm, rotated rx 180 ry 0 rz 0.01 deg; joints [26.547, -44.147, 102.435, -149.744, 62.552, 166.021]
  MoveC 2948 to (-316.8, -17.95, -30) mm, rotated rx -180 ry 0 rz 0.01 deg; joints [26.432, -44.142, 102.429, -149.869, 62.521, 166.079] to (-318.31, -20.59, -30) mm, rotated rx 180 ry 0 rz 0.01 deg; joints [26.318, -44.131, 102.412, -149.992, 62.485, 166.134]
  MoveC 2949 to (-318.33, -22.81, -30) mm, rotated rx 180 ry 0 rz 0.01 deg; joints [26.242, -44.172, 102.502, -150.087, 62.509, 166.201] to (-316.42, -23.92, -30) mm, rotated rx 180 ry 0 rz 0.01 deg; joints [26.236, -44.268, 102.711, -150.122, 62.604, 166.267]
  MoveL 2950 to (-77.12, -23.92, -30) mm, rotated rx -180 ry 0 rz 0.01 deg; joints [30.9, -52.774, 121.161, -147.343, 72.185, 169.915]
  MoveC 2951 to (-75.19, -22.81, -30) mm, rotated rx 180 ry 0 rz 0.01 deg; joints [30.986, -52.816, 121.251, -147.263, 72.243, 169.914] to (-75.19, -20.57, -30) mm, rotated rx -180 ry 0 rz 0.01 deg; joints [31.07, -52.776, 121.156, -147.167, 72.214, 169.856]
  MoveC 2952 to (-78.74, -12.56, -30) mm, rotated rx 180 ry 0 rz 0.01 deg; joints [31.29, -52.517, 120.562, -146.882, 71.978, 169.593] to (-80.54, -3.98, -30) mm, rotated rx 180 ry 0 rz 0.01 deg; joints [31.569, -52.301, 120.065, -146.544, 71.8, 169.338]
  MoveC 2953 to (-80.32, 4.81, -30) mm, rotated rx 180 ry 0 rz 0.01 deg; joints [31.899, -52.144, 119.697, -146.165, 71.694, 169.105] to (-77.93, 13.27, -30) mm, rotated rx 180 ry 0 rz 0.01 deg; joints [32.265, -52.06, 119.492, -145.766, 71.672, 168.911]
  MoveL 2954 to (-57.47, 49.9, -30) mm, rotated rx -180 ry 0 rz 0.01 deg; joints [34.078, -51.987, 119.251, -143.874, 71.937, 168.208]
  MoveC 2955 to (-51.32, 57.8, -30) mm, rotated rx -180 ry 0 rz 0.01 deg; joints [34.511, -52.019, 119.304, -143.435, 72.053, 168.08] to (-43.25, 63.74, -30) mm, rotated rx -180 ry 0 rz 0.01 deg; joints [34.922, -52.148, 119.576, -143.043, 72.262, 168.037]
  MoveC 2956 to (-34.02, 67.54, -30) mm, rotated rx -180 ry 0 rz 0.01 deg; joints [35.288, -52.354, 120.022, -142.715, 72.538, 168.072] to (-24.21, 69.35, -30) mm, rotated rx -180 ry 0 rz 0.01 deg; joints [35.601, -52.616, 120.598, -142.456, 72.859, 168.173]
  MoveC 2957 to (-18.88, 69.28, -30) mm, rotated rx 180 ry 0 rz 0.01 deg; joints [35.734, -52.779, 120.96, -142.356, 73.047, 168.259] to (-13.66, 68.24, -30) mm, rotated rx 180 ry 0 rz 0.01 deg; joints [35.832, -52.958, 121.359, -142.298, 73.243, 168.37]
  MoveC 2958 to (-8.66, 66.42, -30) mm, rotated rx -180 ry 0 rz 0.01 deg; joints [35.896, -53.146, 121.78, -142.275, 73.442, 168.499] to (-3.94, 63.97, -30) mm, rotated rx 180 ry 0 rz 0.01 deg; joints [35.931, -53.337, 122.211, -142.283, 73.64, 168.642]
  MoveC 2959 to (-2.95, 63.3, -30) mm, rotated rx 180 ry 0 rz 0.01 deg; joints [35.932, -53.381, 122.309, -142.292, 73.683, 168.676] to (-2.05, 62.52, -30) mm, rotated rx 180 ry 0 rz 0.01 deg; joints [35.928, -53.424, 122.407, -142.306, 73.725, 168.712]
  MoveC 2960 to (-1.17, 61.71, -30) mm, rotated rx 180 ry 0 rz 0.01 deg; joints [35.922, -53.466, 122.504, -142.322, 73.767, 168.749] to (-0.26, 60.94, -30) mm, rotated rx 180 ry 0 rz 0.01 deg; joints [35.918, -53.509, 122.601, -142.335, 73.809, 168.784]
  MoveC 2961 to (1.82, 60.7, -30) mm, rotated rx 180 ry 0 rz 0.01 deg; joints [35.964, -53.576, 122.75, -142.304, 73.884, 168.823] to (2.93, 62.47, -30) mm, rotated rx -180 ry 0 rz 0.01 deg; joints [36.057, -53.572, 122.739, -142.208, 73.898, 168.791]
  MoveL 2962 to (2.92, 328.01, -30) mm, rotated rx -180 ry 0 rz 0.01 deg; joints [44.546, -47.041, 108.005, -131.838, 70.346, 160.18]
  MoveC 2963 to (1.79, 330.74, -30) mm, rotated rx -180 ry 0 rz 0.01 deg; joints [44.591, -46.928, 107.76, -131.758, 70.274, 160.06] to (-0.93, 331.87, -30) mm, rotated rx -180 ry 0 rz 0.01 deg; joints [44.548, -46.813, 107.513, -131.766, 70.17, 159.97]
  MoveL 2964 to (-150.1, 331.86, -30) mm, rotated rx -180 ry 0 rz 0.01 deg; joints [40.724, -41.93, 97.146, -133.92, 64.954, 157.115]
  MoveC 2965 to (-151.73, 330.79, -30) mm, rotated rx 180 ry 0 rz 0.01 deg; joints [40.656, -41.904, 97.092, -133.979, 64.907, 157.123] to (-151.4, 328.87, -30) mm, rotated rx 180 ry 0 rz 0.01 deg; joints [40.61, -41.973, 97.241, -134.052, 64.943, 157.206]
  MoveC 2966 to (-143.85, 317.77, -30) mm, rotated rx 180 ry 0 rz 0.01 deg; joints [40.481, -42.567, 98.51, -134.406, 65.362, 157.796] to (-139.99, 304.93, -30) mm, rotated rx 180 ry 0 rz 0.01 deg; joints [40.212, -43.076, 99.603, -134.868, 65.667, 158.369]
  MoveC 2967 to (-140.28, 291.49, -30) mm, rotated rx -180 ry 0 rz 0.01 deg; joints [39.822, -43.448, 100.413, -135.4, 65.825, 158.872] to (-144.82, 278.85, -30) mm, rotated rx -180 ry 0 rz 0.01 deg; joints [39.35, -43.645, 100.848, -135.954, 65.817, 159.257]
  MoveC 2968 to (-150.77, 271.07, -30) mm, rotated rx -180 ry 0 rz 0.01 deg; joints [38.984, -43.653, 100.877, -136.333, 65.695, 159.43] to (-158.71, 265.33, -30) mm, rotated rx -180 ry 0 rz 0.01 deg; joints [38.63, -43.531, 100.628, -136.653, 65.471, 159.486]
  MoveC 2969 to (-167.7, 261.63, -30) mm, rotated rx 180 ry 0 rz 0.01 deg; joints [38.313, -43.313, 100.173, -136.902, 65.179, 159.446] to (-177.21, 259.57, -30) mm, rotated rx -180 ry 0 rz 0.01 deg; joints [38.035, -43.029, 99.576, -137.088, 64.846, 159.333]
  MoveL 2970 to (-214.9, 259.48, -30) mm, rotated rx -180 ry 0 rz 0.01 deg; joints [37.187, -41.646, 96.658, -137.453, 63.394, 158.565]
  MoveC 2971 to (-224.72, 260.81, -30) mm, rotated rx -180 ry 0 rz 0.01 deg; joints [37.011, -41.239, 95.797, -137.481, 62.992, 158.306] to (-233.83, 264.71, -30) mm, rotated rx 180 ry 0 rz 0.01 deg; joints [36.925, -40.782, 94.83, -137.391, 62.583, 157.959]
  MoveC 2972 to (-241.73, 270.64, -30) mm, rotated rx -180 ry 0 rz 0.01 deg; joints [36.925, -40.309, 93.829, -137.204, 62.194, 157.554] to (-248.22, 278.08, -30) mm, rotated rx -180 ry 0 rz 0.01 deg; joints [36.998, -39.843, 92.84, -136.939, 61.841, 157.115]
  MoveC 2973 to (-250.52, 282.11, -30) mm, rotated rx 180 ry 0 rz 0.01 deg; joints [37.063, -39.636, 92.399, -136.786, 61.697, 156.901] to (-252.04, 286.51, -30) mm, rotated rx 180 ry 0 rz 0.01 deg; joints [37.155, -39.449, 92, -136.613, 61.581, 156.69]
  MoveC 2974 to (-253.11, 291.01, -30) mm, rotated rx 180 ry 0 rz 0.01 deg; joints [37.258, -39.275, 91.629, -136.432, 61.482, 156.484] to (-254.14, 295.52, -30) mm, rotated rx -180 ry 0 rz 0.01 deg; joints [37.363, -39.101, 91.258, -136.251, 61.383, 156.276]
  MoveC 2975 to (-254.54, 299.22, -30) mm, rotated rx -180 ry 0 rz 0.01 deg; joints [37.458, -38.975, 90.989, -136.099, 61.32, 156.115] to (-254.12, 302.93, -30) mm, rotated rx -180 ry 0 rz 0.01 deg; joints [37.57, -38.881, 90.787, -135.942, 61.291, 155.973]
  MoveC 2976 to (-253.37, 306.55, -30) mm, rotated rx -180 ry 0 rz 0.01 deg; joints [37.687, -38.803, 90.618, -135.787, 61.276, 155.842] to (-252.74, 310.2, -30) mm, rotated rx -180 ry 0 rz 0.01 deg; joints [37.801, -38.718, 90.435, -135.632, 61.255, 155.706]
  MoveC 2977 to (-251.35, 315.36, -30) mm, rotated rx -180 ry 0 rz 0.01 deg; joints [37.974, -38.617, 90.216, -135.409, 61.246, 155.525] to (-248.87, 320.09, -30) mm, rotated rx -180 ry 0 rz 0.01 deg; joints [38.158, -38.572, 90.115, -135.199, 61.287, 155.387]
  MoveC 2978 to (-247.39, 322.21, -30) mm, rotated rx 180 ry 0 rz 0.01 deg; joints [38.248, -38.566, 90.1, -135.103, 61.319, 155.334] to (-245.85, 324.29, -30) mm, rotated rx 180 ry 0 rz 0.01 deg; joints [38.338, -38.563, 90.091, -135.008, 61.355, 155.284]
  MoveL 2979 to (-245.68, 324.89, -29.83) mm, rotated rx 180 ry 0 rz 0.01 deg; joints [38.359, -38.559, 90.066, -134.979, 61.349, 155.257]
  MoveL 2980 to (-245.75, 325.35, -29.37) mm, rotated rx 180 ry 0 rz 0.01 deg; joints [38.369, -38.564, 90.032, -134.953, 61.326, 155.22]
  MoveL 2981 to (-245.82, 325.51, -28.73) mm, rotated rx 180 ry 0 rz 0.01 deg; joints [38.372, -38.586, 90.019, -134.937, 61.303, 155.191]
  Set speed (500.0 mm/s)
  MoveL 2982 to (-245.82, 325.51, 11) mm, rotated rx 180 ry 0 rz 0.01 deg; joints [38.355, -40.402, 90.12, -134.269, 60.091, 153.8]
  Set speed (500.0 mm/s)
  MoveL 2983 to (-398.5, 339.2, 11) mm, rotated rx -180 ry 0 rz 0.01 deg; joints [35.632, -33.026, 75.127, -133.489, 53.441, 148.81]
  Set speed (100.0 mm/s)
  MoveL 2984 to (-398.5, 339.2, -8.23) mm, rotated rx -180 ry 0 rz 0.01 deg; joints [35.64, -32.232, 75.091, -133.883, 53.969, 149.485]
  MoveL 2985 to (-398.51, 339.2, -8.36) mm, rotated rx -180 ry 0 rz 0.01 deg; joints [35.64, -32.226, 75.09, -133.886, 53.972, 149.49]
  MoveL 2986 to (-398.77, 339.19, -9.01) mm, rotated rx -180 ry 0 rz 0.01 deg; joints [35.636, -32.186, 75.062, -133.897, 53.978, 149.503]
  MoveL 2987 to (-399.34, 339.13, -9.43) mm, rotated rx -180 ry 0 rz 0.01 deg; joints [35.623, -32.142, 75.007, -133.904, 53.964, 149.5]
  MoveL 2988 to (-399.69, 339.08, -9.5) mm, rotated rx -180 ry 0 rz 0.01 deg; joints [35.615, -32.123, 74.974, -133.905, 53.95, 149.493]
  MoveL 2989 to (-399.72, 339.07, -9.5) mm, rotated rx -180 ry 0 rz 0.01 deg; joints [35.615, -32.122, 74.971, -133.905, 53.949, 149.493]
  MoveL 2990 to (-400.55, 338.85, -9.53) mm, rotated rx -180 ry 0 rz 0.01 deg; joints [35.593, -32.087, 74.902, -133.91, 53.914, 149.476]
  MoveL 2991 to (-400.6, 338.83, -9.53) mm, rotated rx 180 ry 0 rz 0.01 deg; joints [35.592, -32.085, 74.899, -133.91, 53.912, 149.475]
  MoveL 2992 to (-401.28, 338.49, -9.56) mm, rotated rx -180 ry 0 rz 0.01 deg; joints [35.57, -32.061, 74.853, -133.922, 53.885, 149.469]
  MoveL 2993 to (-401.4, 338.42, -9.56) mm, rotated rx 180 ry 0 rz 0.01 deg; joints [35.566, -32.057, 74.845, -133.924, 53.88, 149.469]
  MoveL 2994 to (-402.84, 337.05, -9.63) mm, rotated rx -180 ry 0 rz 0.01 deg; joints [35.503, -32.03, 74.797, -133.979, 53.832, 149.49]
  MoveL 2995 to (-402.87, 337.02, -9.63) mm, rotated rx -180 ry 0 rz 0.01 deg; joints [35.501, -32.03, 74.797, -133.981, 53.832, 149.491]
  MoveL 2996 to (-403.75, 334.43, -9.73) mm, rotated rx 180 ry 0 rz 0.01 deg; joints [35.417, -32.073, 74.896, -134.1, 53.826, 149.594]
  MoveL 2997 to (-403.78, 333.95, -9.75) mm, rotated rx 180 ry 0 rz 0.01 deg; joints [35.403, -32.088, 74.929, -134.123, 53.831, 149.618]
  MoveL 2998 to (-403.79, 333.65, -9.76) mm, rotated rx -180 ry 0 rz 0.01 deg; joints [35.395, -32.097, 74.949, -134.137, 53.835, 149.633]
  MoveL 2999 to (-403.79, 333.05, -9.78) mm, rotated rx -180 ry 0 rz 0.01 deg; joints [35.38, -32.118, 74.994, -134.166, 53.843, 149.665]
  MoveL 3000 to (-401.25, 328.08, -9.98) mm, rotated rx 180 ry 0 rz 0.01 deg; joints [35.296, -32.411, 75.617, -134.427, 54.03, 150.01]
  MoveL 3001 to (-395.74, 327.2, -10.18) mm, rotated rx -180 ry 0 rz 0.01 deg; joints [35.376, -32.708, 76.243, -134.512, 54.303, 150.249]
  MoveL 3002 to (-391.79, 331.15, -10.39) mm, rotated rx 180 ry 0 rz 0.01 deg; joints [35.556, -32.758, 76.358, -134.356, 54.44, 150.194]
  MoveL 3003 to (-392.66, 336.66, -10.59) mm, rotated rx -180 ry 0 rz 0.01 deg; joints [35.685, -32.514, 75.868, -134.093, 54.336, 149.896]
  MoveL 3004 to (-397.64, 339.2, -10.79) mm, rotated rx 180 ry 0 rz 0.01 deg; joints [35.658, -32.168, 75.172, -133.941, 54.079, 149.603]
  MoveL 3005 to (-398.51, 339.2, -10.82) mm, rotated rx -180 ry 0 rz 0.01 deg; joints [35.641, -32.123, 75.083, -133.935, 54.039, 149.574]
  MoveL 3006 to (-399.34, 339.13, -10.85) mm, rotated rx -180 ry 0 rz 0.01 deg; joints [35.624, -32.083, 75.002, -133.932, 54.002, 149.549]
  MoveL 3007 to (-399.69, 339.08, -10.86) mm, rotated rx -180 ry 0 rz 0.01 deg; joints [35.616, -32.066, 74.97, -133.932, 53.987, 149.54]
  MoveL 3008 to (-400.55, 338.85, -10.89) mm, rotated rx 180 ry 0 rz 0.01 deg; joints [35.594, -32.03, 74.898, -133.937, 53.951, 149.523]
  MoveL 3009 to (-400.6, 338.83, -10.9) mm, rotated rx -180 ry 0 rz 0.01 deg; joints [35.592, -32.028, 74.895, -133.937, 53.949, 149.522]
  MoveL 3010 to (-401.28, 338.49, -10.92) mm, rotated rx -180 ry 0 rz 0.01 deg; joints [35.571, -32.004, 74.849, -133.949, 53.922, 149.516]
  MoveL 3011 to (-401.4, 338.42, -10.93) mm, rotated rx -180 ry 0 rz 0.01 deg; joints [35.566, -32, 74.842, -133.951, 53.917, 149.516]
  MoveL 3012 to (-402.84, 337.05, -11) mm, rotated rx -180 ry 0 rz 0.01 deg; joints [35.503, -31.973, 74.793, -134.007, 53.87, 149.537]
  MoveL 3013 to (-402.87, 337.02, -11) mm, rotated rx -180 ry 0 rz 0.01 deg; joints [35.502, -31.973, 74.793, -134.008, 53.869, 149.538]
  MoveL 3014 to (-403.75, 334.43, -11.1) mm, rotated rx -180 ry 0 rz 0.01 deg; joints [35.417, -32.016, 74.892, -134.127, 53.863, 149.641]
  MoveL 3015 to (-403.78, 333.95, -11.11) mm, rotated rx -180 ry 0 rz 0.01 deg; joints [35.404, -32.031, 74.925, -134.15, 53.869, 149.665]
  MoveL 3016 to (-403.79, 333.65, -11.12) mm, rotated rx -180 ry 0 rz 0.01 deg; joints [35.396, -32.04, 74.945, -134.164, 53.872, 149.68]
  MoveL 3017 to (-403.79, 333.05, -11.14) mm, rotated rx -180 ry 0 rz 0.01 deg; joints [35.38, -32.061, 74.99, -134.194, 53.881, 149.711]
  MoveL 3018 to (-401.25, 328.08, -11.35) mm, rotated rx 180 ry 0 rz 0.01 deg; joints [35.296, -32.354, 75.613, -134.454, 54.068, 150.057]
  MoveL 3019 to (-395.74, 327.2, -11.55) mm, rotated rx 180 ry 0 rz 0.01 deg; joints [35.377, -32.65, 76.239, -134.538, 54.34, 150.296]
  MoveL 3020 to (-391.79, 331.15, -11.75) mm, rotated rx 180 ry 0 rz 0.01 deg; joints [35.556, -32.701, 76.354, -134.382, 54.478, 150.24]
  MoveL 3021 to (-392.66, 336.66, -11.95) mm, rotated rx -180 ry 0 rz 0.01 deg; joints [35.686, -32.457, 75.864, -134.12, 54.373, 149.943]
  MoveL 3022 to (-397.64, 339.2, -12.16) mm, rotated rx -180 ry 0 rz 0.01 deg; joints [35.658, -32.111, 75.168, -133.968, 54.116, 149.65]
  MoveL 3023 to (-398.51, 339.2, -12.19) mm, rotated rx -180 ry 0 rz 0.01 deg; joints [35.642, -32.066, 75.079, -133.962, 54.076, 149.621]
  MoveL 3024 to (-399.34, 339.13, -12.22) mm, rotated rx 180 ry 0 rz 0.01 deg; joints [35.625, -32.026, 74.998, -133.959, 54.04, 149.596]
  MoveL 3025 to (-399.69, 339.08, -12.23) mm, rotated rx -180 ry 0 rz 0.01 deg; joints [35.616, -32.009, 74.966, -133.959, 54.024, 149.587]
  MoveL 3026 to (-400.55, 338.85, -12.26) mm, rotated rx -180 ry 0 rz 0.01 deg; joints [35.594, -31.973, 74.894, -133.964, 53.988, 149.569]
  MoveL 3027 to (-400.6, 338.83, -12.26) mm, rotated rx 180 ry 0 rz 0.01 deg; joints [35.593, -31.971, 74.89, -133.965, 53.986, 149.569]
  MoveL 3028 to (-401.28, 338.49, -12.29) mm, rotated rx -180 ry 0 rz 0.01 deg; joints [35.571, -31.947, 74.844, -133.976, 53.959, 149.563]
  MoveL 3029 to (-401.4, 338.42, -12.29) mm, rotated rx -180 ry 0 rz 0.01 deg; joints [35.567, -31.943, 74.837, -133.979, 53.954, 149.562]
  MoveL 3030 to (-402.84, 337.05, -12.36) mm, rotated rx -180 ry 0 rz 0.01 deg; joints [35.504, -31.916, 74.789, -134.034, 53.907, 149.583]
  MoveL 3031 to (-402.87, 337.02, -12.36) mm, rotated rx 180 ry 0 rz 0.01 deg; joints [35.503, -31.916, 74.789, -134.035, 53.906, 149.584]
  MoveL 3032 to (-403.75, 334.43, -12.46) mm, rotated rx -180 ry 0 rz 0.01 deg; joints [35.418, -31.959, 74.888, -134.154, 53.9, 149.688]
  MoveL 3033 to (-403.78, 333.95, -12.48) mm, rotated rx -180 ry 0 rz 0.01 deg; joints [35.405, -31.974, 74.921, -134.177, 53.906, 149.712]
  MoveL 3034 to (-403.79, 333.65, -12.49) mm, rotated rx 180 ry 0 rz 0.01 deg; joints [35.397, -31.983, 74.941, -134.191, 53.91, 149.727]
  MoveL 3035 to (-403.79, 333.05, -12.51) mm, rotated rx -180 ry 0 rz 0.01 deg; joints [35.381, -32.003, 74.986, -134.221, 53.918, 149.758]
  MoveL 3036 to (-401.25, 328.08, -12.71) mm, rotated rx 180 ry 0 rz 0.01 deg; joints [35.297, -32.296, 75.609, -134.481, 54.105, 150.103]
  MoveL 3037 to (-395.74, 327.2, -12.91) mm, rotated rx 180 ry 0 rz 0.01 deg; joints [35.377, -32.593, 76.235, -134.565, 54.378, 150.342]
  MoveL 3038 to (-391.79, 331.15, -13.12) mm, rotated rx 180 ry 0 rz 0.01 deg; joints [35.557, -32.643, 76.35, -134.409, 54.516, 150.287]
  MoveL 3039 to (-392.66, 336.66, -13.32) mm, rotated rx -180 ry 0 rz 0.01 deg; joints [35.686, -32.399, 75.86, -134.147, 54.411, 149.989]
  MoveL 3040 to (-397.64, 339.2, -13.52) mm, rotated rx -180 ry 0 rz 0.01 deg; joints [35.659, -32.054, 75.164, -133.995, 54.153, 149.697]
  MoveL 3041 to (-398.51, 339.2, -13.55) mm, rotated rx 180 ry 0 rz 0.01 deg; joints [35.643, -32.009, 75.075, -133.989, 54.114, 149.668]
  MoveL 3042 to (-399.34, 339.13, -13.58) mm, rotated rx -180 ry 0 rz 0.01 deg; joints [35.625, -31.968, 74.994, -133.986, 54.077, 149.643]
  MoveL 3043 to (-399.69, 339.08, -13.59) mm, rotated rx -180 ry 0 rz 0.01 deg; joints [35.617, -31.952, 74.961, -133.986, 54.061, 149.634]
  MoveL 3044 to (-400.55, 338.85, -13.62) mm, rotated rx 180 ry 0 rz 0.01 deg; joints [35.595, -31.915, 74.889, -133.991, 54.025, 149.616]
  MoveL 3045 to (-400.6, 338.83, -13.63) mm, rotated rx -180 ry 0 rz 0.01 deg; joints [35.594, -31.914, 74.886, -133.992, 54.023, 149.615]
  MoveL 3046 to (-401.28, 338.49, -13.65) mm, rotated rx 180 ry 0 rz 0.01 deg; joints [35.572, -31.89, 74.84, -134.003, 53.996, 149.609]
  MoveL 3047 to (-401.4, 338.42, -13.66) mm, rotated rx 180 ry 0 rz 0.01 deg; joints [35.567, -31.886, 74.833, -134.006, 53.991, 149.609]
  MoveL 3048 to (-402.84, 337.05, -13.73) mm, rotated rx -180 ry 0 rz 0.01 deg; joints [35.505, -31.859, 74.785, -134.061, 53.944, 149.63]
  MoveL 3049 to (-402.87, 337.02, -13.73) mm, rotated rx -180 ry 0 rz 0.01 deg; joints [35.503, -31.859, 74.785, -134.062, 53.943, 149.631]
  MoveL 3050 to (-403.75, 334.43, -13.83) mm, rotated rx -180 ry 0 rz 0.01 deg; joints [35.418, -31.901, 74.883, -134.181, 53.937, 149.734]
  MoveL 3051 to (-403.78, 333.95, -13.84) mm, rotated rx -180 ry 0 rz 0.01 deg; joints [35.405, -31.916, 74.916, -134.204, 53.943, 149.758]
  MoveL 3052 to (-403.79, 333.65, -13.85) mm, rotated rx 180 ry 0 rz 0.01 deg; joints [35.397, -31.926, 74.937, -134.218, 53.947, 149.773]
  MoveL 3053 to (-403.79, 333.05, -13.87) mm, rotated rx -180 ry 0 rz 0.01 deg; joints [35.381, -31.946, 74.981, -134.248, 53.955, 149.804]
  MoveL 3054 to (-401.25, 328.08, -14.08) mm, rotated rx 180 ry 0 rz 0.01 deg; joints [35.297, -32.239, 75.605, -134.508, 54.143, 150.15]
  MoveL 3055 to (-395.74, 327.2, -14.28) mm, rotated rx 180 ry 0 rz 0.01 deg; joints [35.378, -32.535, 76.231, -134.591, 54.416, 150.388]
  MoveL 3056 to (-391.79, 331.15, -14.48) mm, rotated rx -180 ry 0 rz 0.01 deg; joints [35.557, -32.585, 76.345, -134.435, 54.553, 150.333]
  MoveL 3057 to (-392.66, 336.66, -14.68) mm, rotated rx -180 ry 0 rz 0.01 deg; joints [35.687, -32.342, 75.855, -134.173, 54.448, 150.036]
  MoveL 3058 to (-397.64, 339.2, -14.89) mm, rotated rx 180 ry 0 rz 0.01 deg; joints [35.66, -31.996, 75.16, -134.022, 54.19, 149.743]
  MoveL 3059 to (-398.51, 339.2, -14.92) mm, rotated rx -180 ry 0 rz 0.01 deg; joints [35.643, -31.952, 75.07, -134.016, 54.151, 149.714]
  MoveL 3060 to (-399.34, 339.13, -14.94) mm, rotated rx 180 ry 0 rz 0.01 deg; joints [35.626, -31.911, 74.99, -134.013, 54.114, 149.689]
  MoveL 3061 to (-399.69, 339.08, -14.96) mm, rotated rx -180 ry 0 rz 0.01 deg; joints [35.618, -31.895, 74.957, -134.013, 54.098, 149.68]
  MoveL 3062 to (-400.55, 338.85, -14.99) mm, rotated rx 180 ry 0 rz 0.01 deg; joints [35.595, -31.858, 74.885, -134.018, 54.062, 149.663]
  MoveL 3063 to (-400.6, 338.83, -14.99) mm, rotated rx -180 ry 0 rz 0.01 deg; joints [35.594, -31.857, 74.882, -134.018, 54.06, 149.662]
  MoveL 3064 to (-401.28, 338.49, -15.02) mm, rotated rx -180 ry 0 rz 0.01 deg; joints [35.572, -31.833, 74.836, -134.03, 54.033, 149.656]
  MoveL 3065 to (-401.4, 338.42, -15.02) mm, rotated rx -180 ry 0 rz 0.01 deg; joints [35.568, -31.829, 74.829, -134.033, 54.028, 149.655]
  MoveL 3066 to (-402.84, 337.05, -15.09) mm, rotated rx -180 ry 0 rz 0.01 deg; joints [35.505, -31.802, 74.78, -134.088, 53.981, 149.676]
  MoveL 3067 to (-402.87, 337.02, -15.09) mm, rotated rx 180 ry 0 rz 0.01 deg; joints [35.504, -31.802, 74.78, -134.089, 53.98, 149.677]
  MoveL 3068 to (-403.75, 334.43, -15.19) mm, rotated rx -180 ry 0 rz 0.01 deg; joints [35.419, -31.844, 74.879, -134.208, 53.975, 149.781]
  MoveL 3069 to (-403.78, 333.95, -15.21) mm, rotated rx 180 ry 0 rz 0.01 deg; joints [35.406, -31.859, 74.912, -134.231, 53.98, 149.805]
  MoveL 3070 to (-403.79, 333.65, -15.22) mm, rotated rx -180 ry 0 rz 0.01 deg; joints [35.398, -31.869, 74.933, -134.245, 53.984, 149.82]
  MoveL 3071 to (-403.79, 333.05, -15.24) mm, rotated rx -180 ry 0 rz 0.01 deg; joints [35.382, -31.889, 74.977, -134.274, 53.992, 149.851]
  MoveL 3072 to (-401.25, 328.08, -15.44) mm, rotated rx -180 ry 0 rz 0.01 deg; joints [35.298, -32.181, 75.6, -134.534, 54.18, 150.196]
  MoveL 3073 to (-395.74, 327.2, -15.64) mm, rotated rx 180 ry 0 rz 0.01 deg; joints [35.379, -32.477, 76.226, -134.618, 54.453, 150.435]
  MoveL 3074 to (-391.79, 331.15, -15.85) mm, rotated rx -180 ry 0 rz 0.01 deg; joints [35.558, -32.528, 76.341, -134.462, 54.591, 150.379]
  MoveL 3075 to (-392.66, 336.66, -16.05) mm, rotated rx -180 ry 0 rz 0.01 deg; joints [35.687, -32.284, 75.851, -134.2, 54.485, 150.082]
  MoveL 3076 to (-397.64, 339.2, -16.25) mm, rotated rx -180 ry 0 rz 0.01 deg; joints [35.66, -31.939, 75.155, -134.048, 54.227, 149.79]
  MoveL 3077 to (-398.51, 339.2, -16.28) mm, rotated rx -180 ry 0 rz 0.01 deg; joints [35.644, -31.894, 75.066, -134.042, 54.187, 149.76]
  MoveL 3078 to (-399.34, 339.13, -16.31) mm, rotated rx 180 ry 0 rz 0.01 deg; joints [35.626, -31.854, 74.985, -134.04, 54.15, 149.736]
  MoveL 3079 to (-399.69, 339.08, -16.32) mm, rotated rx -180 ry 0 rz 0.01 deg; joints [35.618, -31.837, 74.952, -134.04, 54.135, 149.727]
  MoveL 3080 to (-400.55, 338.85, -16.35) mm, rotated rx 180 ry 0 rz 0.01 deg; joints [35.596, -31.801, 74.88, -134.045, 54.099, 149.709]
  MoveL 3081 to (-400.6, 338.83, -16.35) mm, rotated rx 180 ry 0 rz 0.01 deg; joints [35.595, -31.799, 74.877, -134.045, 54.097, 149.708]
  MoveL 3082 to (-401.28, 338.49, -16.38) mm, rotated rx -180 ry 0 rz 0.01 deg; joints [35.573, -31.776, 74.831, -134.057, 54.07, 149.702]
  MoveL 3083 to (-401.4, 338.42, -16.39) mm, rotated rx -180 ry 0 rz 0.01 deg; joints [35.569, -31.772, 74.824, -134.059, 54.065, 149.702]
  MoveL 3084 to (-402.84, 337.05, -16.46) mm, rotated rx 180 ry 0 rz 0.01 deg; joints [35.506, -31.745, 74.776, -134.115, 54.018, 149.723]
  MoveL 3085 to (-402.87, 337.02, -16.46) mm, rotated rx 180 ry 0 rz 0.01 deg; joints [35.504, -31.745, 74.776, -134.116, 54.017, 149.724]
  MoveL 3086 to (-403.75, 334.43, -16.55) mm, rotated rx 180 ry 0 rz 0.01 deg; joints [35.42, -31.787, 74.874, -134.235, 54.012, 149.827]
  MoveL 3087 to (-403.78, 333.95, -16.57) mm, rotated rx 180 ry 0 rz 0.01 deg; joints [35.406, -31.802, 74.907, -134.258, 54.017, 149.851]
  MoveL 3088 to (-403.79, 333.65, -16.58) mm, rotated rx -180 ry 0 rz 0.01 deg; joints [35.398, -31.811, 74.928, -134.272, 54.021, 149.866]
  MoveL 3089 to (-403.79, 333.05, -16.6) mm, rotated rx 180 ry 0 rz 0.01 deg; joints [35.383, -31.832, 74.972, -134.301, 54.029, 149.897]
  MoveL 3090 to (-401.25, 328.08, -16.8) mm, rotated rx 180 ry 0 rz 0.01 deg; joints [35.299, -32.124, 75.596, -134.561, 54.218, 150.242]
  MoveL 3091 to (-395.74, 327.2, -17.01) mm, rotated rx -180 ry 0 rz 0.01 deg; joints [35.379, -32.42, 76.221, -134.644, 54.491, 150.481]
  MoveL 3092 to (-391.79, 331.15, -17.21) mm, rotated rx -180 ry 0 rz 0.01 deg; joints [35.559, -32.47, 76.336, -134.488, 54.628, 150.425]
  MoveL 3093 to (-392.66, 336.66, -17.41) mm, rotated rx 180 ry 0 rz 0.01 deg; joints [35.688, -32.227, 75.846, -134.226, 54.522, 150.128]
  MoveL 3094 to (-397.64, 339.2, -17.61) mm, rotated rx -180 ry 0 rz 0.01 deg; joints [35.661, -31.882, 75.15, -134.075, 54.264, 149.836]
  MoveL 3095 to (-398.51, 339.2, -17.64) mm, rotated rx 180 ry 0 rz 0.01 deg; joints [35.644, -31.837, 75.061, -134.069, 54.224, 149.807]
  MoveL 3096 to (-399.34, 339.13, -17.67) mm, rotated rx -180 ry 0 rz 0.01 deg; joints [35.627, -31.796, 74.98, -134.066, 54.187, 149.782]
  MoveL 3097 to (-399.69, 339.08, -17.69) mm, rotated rx -180 ry 0 rz 0.01 deg; joints [35.619, -31.78, 74.948, -134.067, 54.172, 149.773]
  MoveL 3098 to (-400.55, 338.85, -17.72) mm, rotated rx -180 ry 0 rz 0.01 deg; joints [35.597, -31.744, 74.875, -134.072, 54.135, 149.755]
  MoveL 3099 to (-400.6, 338.83, -17.72) mm, rotated rx -180 ry 0 rz 0.01 deg; joints [35.595, -31.742, 74.872, -134.072, 54.134, 149.755]
  MoveL 3100 to (-401.28, 338.49, -17.75) mm, rotated rx -180 ry 0 rz 0.01 deg; joints [35.574, -31.718, 74.826, -134.083, 54.107, 149.748]
  MoveL 3101 to (-401.4, 338.42, -17.75) mm, rotated rx -180 ry 0 rz 0.01 deg; joints [35.569, -31.714, 74.819, -134.086, 54.102, 149.748]
  MoveL 3102 to (-402.84, 337.05, -17.82) mm, rotated rx 180 ry 0 rz 0.01 deg; joints [35.506, -31.687, 74.771, -134.141, 54.054, 149.769]
  MoveL 3103 to (-402.87, 337.02, -17.82) mm, rotated rx -180 ry 0 rz 0.01 deg; joints [35.505, -31.687, 74.771, -134.143, 54.054, 149.77]
  MoveL 3104 to (-403.75, 334.43, -17.92) mm, rotated rx -180 ry 0 rz 0.01 deg; joints [35.42, -31.73, 74.869, -134.261, 54.049, 149.873]
  MoveL 3105 to (-403.78, 333.95, -17.94) mm, rotated rx 180 ry 0 rz 0.01 deg; joints [35.407, -31.745, 74.902, -134.285, 54.054, 149.897]
  MoveL 3106 to (-403.79, 333.65, -17.95) mm, rotated rx -180 ry 0 rz 0.01 deg; joints [35.399, -31.754, 74.923, -134.299, 54.058, 149.912]
  MoveL 3107 to (-403.79, 333.05, -17.97) mm, rotated rx 180 ry 0 rz 0.01 deg; joints [35.383, -31.774, 74.967, -134.328, 54.066, 149.943]
  MoveL 3108 to (-401.25, 328.08, -18.17) mm, rotated rx 180 ry 0 rz 0.01 deg; joints [35.299, -32.066, 75.591, -134.587, 54.255, 150.288]
  MoveL 3109 to (-395.74, 327.2, -18.37) mm, rotated rx -180 ry 0 rz 0.01 deg; joints [35.38, -32.362, 76.217, -134.67, 54.528, 150.526]
  MoveL 3110 to (-391.79, 331.15, -18.57) mm, rotated rx -180 ry 0 rz 0.01 deg; joints [35.559, -32.412, 76.331, -134.514, 54.666, 150.471]
  MoveL 3111 to (-392.66, 336.66, -18.78) mm, rotated rx -180 ry 0 rz 0.01 deg; joints [35.689, -32.169, 75.841, -134.253, 54.56, 150.175]
  MoveL 3112 to (-397.64, 339.2, -18.98) mm, rotated rx -180 ry 0 rz 0.01 deg; joints [35.661, -31.824, 75.145, -134.102, 54.301, 149.882]
  MoveL 3113 to (-398.51, 339.2, -19.01) mm, rotated rx -180 ry 0 rz 0.01 deg; joints [35.645, -31.779, 75.056, -134.096, 54.261, 149.853]
  MoveL 3114 to (-399.34, 339.13, -19.04) mm, rotated rx 180 ry 0 rz 0.01 deg; joints [35.628, -31.739, 74.975, -134.093, 54.224, 149.828]
  MoveL 3115 to (-399.69, 339.08, -19.05) mm, rotated rx 180 ry 0 rz 0.01 deg; joints [35.619, -31.722, 74.943, -134.093, 54.209, 149.819]
  MoveL 3116 to (-400.55, 338.85, -19.08) mm, rotated rx -180 ry 0 rz 0.01 deg; joints [35.597, -31.686, 74.871, -134.098, 54.172, 149.801]
  MoveL 3117 to (-400.6, 338.83, -19.08) mm, rotated rx -180 ry 0 rz 0.01 deg; joints [35.596, -31.684, 74.867, -134.099, 54.17, 149.801]
  MoveL 3118 to (-401.28, 338.49, -19.11) mm, rotated rx -180 ry 0 rz 0.01 deg; joints [35.574, -31.661, 74.821, -134.11, 54.144, 149.795]
  MoveL 3119 to (-401.4, 338.42, -19.12) mm, rotated rx 180 ry 0 rz 0.01 deg; joints [35.57, -31.657, 74.814, -134.113, 54.139, 149.794]
  MoveL 3120 to (-402.84, 337.05, -19.19) mm, rotated rx -180 ry 0 rz 0.01 deg; joints [35.507, -31.63, 74.766, -134.168, 54.091, 149.815]
  MoveL 3121 to (-402.87, 337.02, -19.19) mm, rotated rx 180 ry 0 rz 0.01 deg; joints [35.506, -31.63, 74.766, -134.169, 54.091, 149.816]
  MoveL 3122 to (-403.75, 334.43, -19.28) mm, rotated rx 180 ry 0 rz 0.01 deg; joints [35.421, -31.672, 74.864, -134.288, 54.086, 149.919]
  MoveL 3123 to (-403.78, 333.95, -19.3) mm, rotated rx 180 ry 0 rz 0.01 deg; joints [35.407, -31.687, 74.897, -134.311, 54.091, 149.943]
  MoveL 3124 to (-403.79, 333.65, -19.31) mm, rotated rx -180 ry 0 rz 0.01 deg; joints [35.4, -31.697, 74.918, -134.325, 54.095, 149.958]
  MoveL 3125 to (-403.79, 333.05, -19.33) mm, rotated rx -180 ry 0 rz 0.01 deg; joints [35.384, -31.717, 74.962, -134.354, 54.103, 149.989]
  MoveL 3126 to (-401.25, 328.08, -19.53) mm, rotated rx -180 ry 0 rz 0.01 deg; joints [35.3, -32.009, 75.586, -134.614, 54.292, 150.334]
  MoveL 3127 to (-395.74, 327.2, -19.74) mm, rotated rx 180 ry 0 rz 0.01 deg; joints [35.38, -32.304, 76.212, -134.697, 54.566, 150.572]
  MoveL 3128 to (-391.79, 331.15, -19.94) mm, rotated rx 180 ry 0 rz 0.01 deg; joints [35.56, -32.354, 76.326, -134.54, 54.703, 150.517]
  MoveL 3129 to (-392.66, 336.66, -20.14) mm, rotated rx 180 ry 0 rz 0.01 deg; joints [35.689, -32.111, 75.836, -134.279, 54.597, 150.221]
  MoveL 3130 to (-397.64, 339.2, -20.34) mm, rotated rx -180 ry 0 rz 0.01 deg; joints [35.662, -31.767, 75.14, -134.128, 54.338, 149.928]
  MoveL 3131 to (-398.51, 339.2, -20.37) mm, rotated rx 180 ry 0 rz 0.01 deg; joints [35.646, -31.722, 75.051, -134.122, 54.298, 149.899]
  MoveL 3132 to (-399.34, 339.13, -20.4) mm, rotated rx 180 ry 0 rz 0.01 deg; joints [35.628, -31.681, 74.97, -134.12, 54.261, 149.874]
  MoveL 3133 to (-399.69, 339.08, -20.42) mm, rotated rx -180 ry 0 rz 0.01 deg; joints [35.62, -31.665, 74.937, -134.12, 54.245, 149.865]
  MoveL 3134 to (-400.55, 338.85, -20.45) mm, rotated rx 180 ry 0 rz 0.01 deg; joints [35.598, -31.629, 74.865, -134.125, 54.209, 149.847]
  MoveL 3135 to (-400.6, 338.83, -20.45) mm, rotated rx -180 ry 0 rz 0.01 deg; joints [35.597, -31.627, 74.862, -134.125, 54.207, 149.847]
  MoveL 3136 to (-401.28, 338.49, -20.47) mm, rotated rx 180 ry 0 rz 0.01 deg; joints [35.575, -31.603, 74.816, -134.137, 54.18, 149.841]
  MoveL 3137 to (-401.4, 338.42, -20.48) mm, rotated rx -180 ry 0 rz 0.01 deg; joints [35.57, -31.599, 74.809, -134.139, 54.176, 149.84]
  MoveL 3138 to (-402.84, 337.05, -20.55) mm, rotated rx -180 ry 0 rz 0.01 deg; joints [35.507, -31.572, 74.761, -134.195, 54.128, 149.861]
  MoveL 3139 to (-402.87, 337.02, -20.55) mm, rotated rx -180 ry 0 rz 0.01 deg; joints [35.506, -31.572, 74.761, -134.196, 54.127, 149.862]
  MoveL 3140 to (-403.75, 334.43, -20.65) mm, rotated rx -180 ry 0 rz 0.01 deg; joints [35.421, -31.615, 74.859, -134.314, 54.122, 149.965]
  MoveL 3141 to (-403.78, 333.95, -20.66) mm, rotated rx -180 ry 0 rz 0.01 deg; joints [35.408, -31.629, 74.892, -134.338, 54.128, 149.989]
  MoveL 3142 to (-403.79, 333.65, -20.68) mm, rotated rx -180 ry 0 rz 0.01 deg; joints [35.4, -31.639, 74.913, -134.352, 54.132, 150.004]
  MoveL 3143 to (-403.79, 333.05, -20.7) mm, rotated rx -180 ry 0 rz 0.01 deg; joints [35.384, -31.659, 74.957, -134.381, 54.14, 150.035]
  MoveL 3144 to (-401.25, 328.08, -20.9) mm, rotated rx 180 ry 0 rz 0.01 deg; joints [35.3, -31.951, 75.581, -134.64, 54.33, 150.379]
  MoveL 3145 to (-395.74, 327.2, -21.1) mm, rotated rx -180 ry 0 rz 0.01 deg; joints [35.381, -32.246, 76.207, -134.723, 54.603, 150.618]
  MoveL 3146 to (-391.79, 331.15, -21.3) mm, rotated rx -180 ry 0 rz 0.01 deg; joints [35.56, -32.296, 76.321, -134.566, 54.741, 150.563]
  MoveL 3147 to (-392.66, 336.66, -21.51) mm, rotated rx -180 ry 0 rz 0.01 deg; joints [35.69, -32.053, 75.831, -134.305, 54.634, 150.266]
  MoveL 3148 to (-397.64, 339.2, -21.71) mm, rotated rx 180 ry 0 rz 0.01 deg; joints [35.662, -31.709, 75.135, -134.154, 54.375, 149.974]
  MoveL 3149 to (-398.51, 339.2, -21.74) mm, rotated rx -180 ry 0 rz 0.01 deg; joints [35.646, -31.664, 75.045, -134.148, 54.335, 149.945]
  MoveL 3150 to (-399.34, 339.13, -21.77) mm, rotated rx -180 ry 0 rz 0.01 deg; joints [35.629, -31.624, 74.965, -134.146, 54.298, 149.92]
  MoveL 3151 to (-399.69, 339.08, -21.78) mm, rotated rx 180 ry 0 rz 0.01 deg; joints [35.621, -31.607, 74.932, -134.146, 54.282, 149.911]
  MoveL 3152 to (-400.55, 338.85, -21.81) mm, rotated rx 180 ry 0 rz 0.01 deg; joints [35.598, -31.571, 74.86, -134.151, 54.246, 149.893]
  MoveL 3153 to (-400.6, 338.83, -21.81) mm, rotated rx 180 ry 0 rz 0.01 deg; joints [35.597, -31.569, 74.857, -134.152, 54.244, 149.893]
  MoveL 3154 to (-401.28, 338.49, -21.84) mm, rotated rx 180 ry 0 rz 0.01 deg; joints [35.575, -31.546, 74.811, -134.163, 54.217, 149.886]
  MoveL 3155 to (-401.4, 338.42, -21.84) mm, rotated rx 180 ry 0 rz 0.01 deg; joints [35.571, -31.542, 74.804, -134.166, 54.212, 149.886]
  MoveL 3156 to (-402.84, 337.05, -21.91) mm, rotated rx -180 ry 0 rz 0.01 deg; joints [35.508, -31.515, 74.755, -134.221, 54.165, 149.907]
  MoveL 3157 to (-402.87, 337.02, -21.92) mm, rotated rx 180 ry 0 rz 0.01 deg; joints [35.507, -31.515, 74.756, -134.223, 54.164, 149.908]
  MoveL 3158 to (-403.75, 334.43, -22.01) mm, rotated rx -180 ry 0 rz 0.01 deg; joints [35.422, -31.557, 74.854, -134.341, 54.159, 150.011]
  MoveL 3159 to (-403.78, 333.95, -22.03) mm, rotated rx 180 ry 0 rz 0.01 deg; joints [35.409, -31.572, 74.887, -134.364, 54.165, 150.035]
  MoveL 3160 to (-403.79, 333.65, -22.04) mm, rotated rx 180 ry 0 rz 0.01 deg; joints [35.401, -31.581, 74.908, -134.378, 54.169, 150.05]
